C03660=1168.556,292.806,-70.556,-176.920,7.929,148.636
C03661=1168.552,293.053,-70.586,-176.917,7.932,148.636
C03662=1168.547,293.302,-70.616,-176.914,7.935,148.636
C03663=1168.544,293.551,-70.646,-176.912,7.938,148.636
C03664=1168.540,293.798,-70.676,-176.909,7.941,148.636
C03665=1168.535,294.047,-70.706,-176.907,7.944,148.636
C03666=1168.531,294.295,-70.736,-176.904,7.947,148.636
C03667=1168.527,294.543,-70.765,-176.902,7.950,148.636
C03668=1168.522,294.791,-70.796,-176.899,7.953,148.636
C03669=1168.518,295.039,-70.826,-176.896,7.956,148.636
C03670=1168.514,295.287,-70.855,-176.894,7.958,148.636
C03671=1168.509,295.535,-70.886,-176.892,7.962,148.636
C03672=1168.505,295.784,-70.915,-176.889,7.965,148.636
C03673=1168.501,296.032,-70.946,-176.886,7.968,148.636
C03674=1168.497,296.281,-70.976,-176.884,7.971,148.637
C03675=1168.493,296.528,-71.006,-176.881,7.974,148.637
C03676=1168.488,296.776,-71.037,-176.878,7.977,148.637
C03677=1168.484,297.024,-71.066,-176.876,7.980,148.637
C03678=1168.480,297.272,-71.097,-176.873,7.983,148.637
C03679=1168.475,297.521,-71.127,-176.871,7.986,148.637
C03680=1168.471,297.769,-71.157,-176.868,7.989,148.637
C03681=1168.467,298.018,-71.187,-176.866,7.992,148.637
C03682=1168.463,298.265,-71.217,-176.863,7.995,148.637
C03683=1168.459,298.513,-71.248,-176.861,7.999,148.637
C03684=1168.455,298.761,-71.278,-176.858,8.002,148.637
C03685=1168.450,299.009,-71.308,-176.855,8.005,148.637
C03686=1168.446,299.257,-71.338,-176.853,8.008,148.637
C03687=1168.442,299.506,-71.369,-176.850,8.011,148.637
C03688=1168.438,299.754,-71.399,-176.847,8.014,148.637
C03689=1168.433,300.002,-71.430,-176.845,8.017,148.637
C03690=1168.429,300.250,-71.461,-176.842,8.020,148.637
C03691=1168.425,300.498,-71.490,-176.840,8.023,148.637
C03692=1168.420,300.747,-71.521,-176.837,8.026,148.637
C03693=1168.417,300.994,-71.551,-176.835,8.029,148.637
C03694=1168.412,301.242,-71.582,-176.832,8.032,148.637
C03695=1168.408,301.490,-71.612,-176.830,8.036,148.637
C03696=1168.403,301.739,-71.642,-176.827,8.039,148.637
C03697=1168.399,301.987,-71.673,-176.825,8.042,148.638
C03698=1168.395,302.235,-71.704,-176.822,8.045,148.638
C03699=1168.391,302.483,-71.734,-176.819,8.048,148.638
C03700=1168.387,302.731,-71.765,-176.817,8.051,148.638
C03701=1168.383,302.979,-71.796,-176.814,8.054,148.638
C03702=1168.378,303.227,-71.826,-176.811,8.057,148.638
C03703=1168.374,303.475,-71.856,-176.809,8.060,148.638
C03704=1168.369,303.723,-71.887,-176.806,8.063,148.638
C03705=1168.365,303.972,-71.918,-176.804,8.067,148.638
C03706=1168.362,304.220,-71.948,-176.801,8.070,148.638
C03707=1168.357,304.468,-71.979,-176.798,8.073,148.638
C03708=1168.352,304.716,-72.009,-176.796,8.076,148.638
C03709=1168.348,304.964,-72.041,-176.793,8.079,148.638
C03710=1168.344,305.212,-72.071,-176.791,8.082,148.638
C03711=1168.340,305.460,-72.102,-176.788,8.085,148.638
C03712=1168.336,305.709,-72.133,-176.786,8.088,148.638
C03713=1168.332,305.956,-72.163,-176.783,8.092,148.639
C03714=1168.327,306.204,-72.194,-176.780,8.095,148.639
C03715=1168.324,306.452,-72.225,-176.778,8.099,148.639
C03716=1168.319,306.700,-72.256,-176.775,8.102,148.639
C03717=1168.314,306.948,-72.287,-176.773,8.105,148.639
C03718=1168.311,307.196,-72.317,-176.770,8.108,148.639
C03719=1168.306,307.444,-72.348,-176.767,8.111,148.639
C03720=1168.302,307.692,-72.379,-176.765,8.114,148.639
C03721=1168.298,307.941,-72.410,-176.762,8.117,148.639
C03722=1168.293,308.189,-72.441,-176.760,8.120,148.639
C03723=1168.290,308.436,-72.472,-176.757,8.123,148.639
C03724=1168.286,308.685,-72.503,-176.755,8.127,148.639
C03725=1168.281,308.933,-72.534,-176.752,8.130,148.639
C03726=1168.276,309.181,-72.564,-176.750,8.133,148.640
C03727=1168.272,309.429,-72.596,-176.747,8.136,148.640
C03728=1168.268,309.677,-72.627,-176.744,8.139,148.639
C03729=1168.264,309.925,-72.658,-176.742,8.142,148.640
C03730=1168.260,310.173,-72.688,-176.739,8.145,148.640
C03731=1168.256,310.420,-72.720,-176.737,8.148,148.640
C03732=1168.252,310.669,-72.751,-176.734,8.151,148.640
C03733=1168.247,310.917,-72.782,-176.732,8.155,148.640
C03734=1168.244,311.165,-72.814,-176.729,8.158,148.640
C03735=1168.239,311.413,-72.844,-176.727,8.161,148.640
C03736=1168.235,311.662,-72.875,-176.724,8.165,148.640
C03737=1168.231,311.909,-72.907,-176.721,8.168,148.640
C03738=1168.226,312.157,-72.938,-176.719,8.171,148.640
C03739=1168.222,312.405,-72.969,-176.716,8.174,148.641
C03740=1168.218,312.653,-73.000,-176.714,8.177,148.641
C03741=1168.214,312.901,-73.031,-176.711,8.181,148.641
C03742=1168.209,313.149,-73.063,-176.709,8.184,148.641
C03743=1168.205,313.397,-73.094,-176.706,8.187,148.641
C03744=1168.201,313.674,-73.129,-176.704,8.190,148.641
C03745=1168.196,313.951,-73.164,-176.701,8.194,148.641
C03746=1168.191,314.228,-73.198,-176.698,8.198,148.641
C03747=1168.187,314.506,-73.234,-176.695,8.201,148.641
C03748=1168.182,314.753,-73.266,-176.692,8.204,148.641
C03749=1168.178,315.002,-73.297,-176.690,8.207,148.642
C03750=1168.174,315.249,-73.328,-176.687,8.210,148.642
C03751=1168.170,315.498,-73.359,-176.685,8.214,148.642
C03752=1168.166,315.745,-73.391,-176.682,8.217,148.642
C03753=1168.162,315.993,-73.423,-176.680,8.221,148.642
C03754=1168.157,316.241,-73.453,-176.677,8.224,148.642
C03755=1168.154,316.489,-73.485,-176.675,8.227,148.642
C03756=1168.149,316.737,-73.516,-176.672,8.230,148.642
C03757=1168.145,316.985,-73.548,-176.670,8.233,148.642
C03758=1168.141,317.232,-73.579,-176.667,8.236,148.642
C03759=1168.136,317.481,-73.611,-176.664,8.240,148.643
C03760=1168.132,317.729,-73.643,-176.662,8.242,148.642
C03761=1168.128,317.977,-73.674,-176.659,8.246,148.643
C03762=1168.125,318.225,-73.706,-176.657,8.249,148.643
C03763=1168.120,318.473,-73.737,-176.654,8.252,148.643
C03764=1168.116,318.721,-73.769,-176.652,8.256,148.643
C03765=1168.111,318.968,-73.801,-176.649,8.259,148.643
C03766=1168.108,319.216,-73.833,-176.647,8.262,148.643
C03767=1168.104,319.465,-73.864,-176.644,8.265,148.643
C03768=1168.099,319.712,-73.895,-176.642,8.269,148.643
C03769=1168.096,319.961,-73.927,-176.639,8.272,148.644
C03770=1168.091,320.208,-73.959,-176.637,8.275,148.644
C03771=1168.087,320.456,-73.991,-176.634,8.278,148.644
C03772=1168.083,320.704,-74.023,-176.631,8.281,148.644
C03773=1168.079,320.952,-74.054,-176.629,8.285,148.644
C03774=1168.074,321.201,-74.086,-176.626,8.289,148.644
C03775=1168.070,321.449,-74.118,-176.624,8.292,148.644
C03776=1168.066,321.696,-74.149,-176.621,8.295,148.644
C03777=1168.062,321.944,-74.181,-176.619,8.298,148.644
C03778=1168.058,322.192,-74.214,-176.616,8.301,148.645
C03779=1168.054,322.440,-74.245,-176.614,8.305,148.645
C03780=1168.050,322.688,-74.277,-176.611,8.308,148.645
C03781=1168.045,322.936,-74.310,-176.609,8.311,148.645
C03782=1168.041,323.183,-74.341,-176.606,8.315,148.645
C03783=1168.037,323.431,-74.373,-176.603,8.318,148.645
C03784=1168.033,323.680,-74.405,-176.601,8.321,148.645
C03785=1168.029,323.927,-74.437,-176.598,8.324,148.645
C03786=1168.025,324.175,-74.469,-176.596,8.327,148.646
C03787=1168.021,324.424,-74.501,-176.594,8.331,148.646
C03788=1168.017,324.672,-74.533,-176.591,8.334,148.646
C03789=1168.013,324.919,-74.564,-176.589,8.337,148.646
C03790=1168.008,325.167,-74.597,-176.586,8.341,148.646
C03791=1168.004,325.415,-74.629,-176.583,8.344,148.646
C03792=1168.000,325.662,-74.661,-176.581,8.347,148.646
C03793=1167.996,325.910,-74.693,-176.579,8.351,148.647
C03794=1167.992,326.158,-74.725,-176.576,8.354,148.647
C03795=1167.988,326.407,-74.758,-176.574,8.357,148.647
C03796=1167.983,326.654,-74.789,-176.571,8.360,148.647
C03797=1167.979,326.902,-74.822,-176.569,8.363,148.647
C03798=1167.976,327.150,-74.854,-176.566,8.367,148.647
C03799=1167.971,327.398,-74.887,-176.563,8.371,148.648
C03800=1167.967,327.646,-74.918,-176.561,8.374,148.648
C03801=1167.962,327.894,-74.950,-176.558,8.377,148.648
C03802=1167.959,328.141,-74.983,-176.556,8.380,148.648
C03803=1167.955,328.390,-75.015,-176.554,8.384,148.648
C03804=1167.951,328.638,-75.047,-176.551,8.387,148.648
C03805=1167.946,328.885,-75.080,-176.548,8.391,148.648
C03806=1167.942,329.133,-75.112,-176.546,8.394,148.649
C03807=1167.938,329.381,-75.144,-176.543,8.397,148.649
C03808=1167.935,329.629,-75.177,-176.541,8.400,148.649
C03809=1167.930,329.877,-75.209,-176.539,8.404,148.649
C03810=1167.926,330.125,-75.242,-176.536,8.407,148.649
C03811=1167.922,330.372,-75.274,-176.533,8.411,148.649
C03812=1167.917,330.620,-75.306,-176.531,8.414,148.649
C03813=1167.914,330.868,-75.338,-176.528,8.417,148.650
C03814=1167.909,331.116,-75.371,-176.526,8.421,148.650
C03815=1167.905,331.364,-75.404,-176.523,8.423,148.650
C03816=1167.902,331.612,-75.436,-176.521,8.427,148.650
C03817=1167.897,331.859,-75.469,-176.518,8.431,148.650
C03818=1167.892,332.107,-75.502,-176.516,8.434,148.650
C03819=1167.889,332.355,-75.534,-176.513,8.437,148.650
C03820=1167.885,332.603,-75.567,-176.511,8.440,148.651
C03821=1167.880,332.851,-75.599,-176.509,8.444,148.651
C03822=1167.877,333.099,-75.632,-176.506,8.447,148.651
C03823=1167.872,333.347,-75.664,-176.504,8.451,148.651
C03824=1167.868,333.595,-75.697,-176.501,8.454,148.651
C03825=1167.864,333.842,-75.729,-176.498,8.457,148.652
C03826=1167.860,334.090,-75.762,-176.496,8.461,148.652
C03827=1167.856,334.338,-75.795,-176.494,8.464,148.652
C03828=1167.852,334.586,-75.827,-176.491,8.468,148.652
C03829=1167.848,334.833,-75.860,-176.488,8.471,148.652
C03830=1167.844,335.081,-75.893,-176.486,8.474,148.652
C03831=1167.839,335.329,-75.926,-176.484,8.478,148.653
C03832=1167.836,335.577,-75.958,-176.481,8.481,148.653
C03833=1167.832,335.825,-75.991,-176.479,8.484,148.653
C03834=1167.827,336.073,-76.024,-176.476,8.488,148.653
C03835=1167.823,336.321,-76.057,-176.474,8.491,148.653
C03836=1167.819,336.568,-76.090,-176.471,8.495,148.653
C03837=1167.815,336.816,-76.123,-176.469,8.498,148.654
C03838=1167.811,337.064,-76.155,-176.467,8.501,148.654
C03839=1167.807,337.312,-76.188,-176.464,8.505,148.654
C03840=1167.803,337.560,-76.221,-176.462,8.509,148.654
C03841=1167.799,337.807,-76.255,-176.459,8.512,148.654
C03842=1167.794,338.055,-76.288,-176.457,8.515,148.655
C03843=1167.791,338.303,-76.320,-176.454,8.518,148.655
C03844=1167.787,338.551,-76.353,-176.451,8.522,148.655
C03845=1167.782,338.799,-76.386,-176.449,8.526,148.655
C03846=1167.778,339.046,-76.419,-176.447,8.529,148.655
C03847=1167.774,339.294,-76.452,-176.445,8.532,148.656
C03848=1167.770,339.574,-76.490,-176.442,8.536,148.656
C03849=1167.764,339.853,-76.527,-176.438,8.540,148.656
C03850=1167.760,340.132,-76.563,-176.435,8.544,148.656
C03851=1167.756,340.412,-76.601,-176.433,8.548,148.656
C03852=1167.751,340.660,-76.634,-176.430,8.552,148.657
C03853=1167.747,340.907,-76.667,-176.428,8.555,148.657
C03854=1167.743,341.155,-76.700,-176.426,8.558,148.657
C03855=1167.739,341.403,-76.733,-176.423,8.562,148.657
C03856=1167.735,341.651,-76.766,-176.421,8.565,148.658
C03857=1167.731,341.898,-76.800,-176.418,8.569,148.658
C03858=1167.727,342.146,-76.833,-176.416,8.572,148.658
C03859=1167.723,342.394,-76.866,-176.414,8.576,148.658
C03860=1167.719,342.641,-76.900,-176.411,8.579,148.658
C03861=1167.715,342.889,-76.933,-176.409,8.583,148.659
C03862=1167.711,343.137,-76.966,-176.406,8.586,148.659
C03863=1167.707,343.385,-77.000,-176.404,8.590,148.659
C03864=1167.703,343.633,-77.033,-176.402,8.593,148.659
C03865=1167.699,343.880,-77.066,-176.399,8.597,148.660
C03866=1167.694,344.128,-77.099,-176.397,8.600,148.660
C03867=1167.690,344.376,-77.133,-176.394,8.604,148.660
C03868=1167.686,344.623,-77.167,-176.392,8.607,148.660
C03869=1167.682,344.871,-77.200,-176.389,8.611,148.660
C03870=1167.678,345.119,-77.233,-176.387,8.614,148.661
C03871=1167.674,345.367,-77.267,-176.385,8.618,148.661
C03872=1167.670,345.615,-77.300,-176.382,8.621,148.661
C03873=1167.666,345.862,-77.334,-176.379,8.625,148.661
C03874=1167.662,346.110,-77.367,-176.377,8.628,148.662
C03875=1167.657,346.358,-77.400,-176.375,8.632,148.662
C03876=1167.653,346.605,-77.434,-176.373,8.635,148.662
C03877=1167.650,346.853,-77.468,-176.370,8.639,148.662
C03878=1167.645,347.101,-77.501,-176.367,8.642,148.662
C03879=1167.641,347.349,-77.534,-176.365,8.646,148.663
C03880=1167.637,347.596,-77.568,-176.362,8.650,148.663
C03881=1167.633,347.844,-77.602,-176.360,8.653,148.663
C03882=1167.629,348.092,-77.636,-176.358,8.656,148.663
C03883=1167.625,348.339,-77.669,-176.355,8.660,148.664
C03884=1167.621,348.587,-77.702,-176.352,8.664,148.664
C03885=1167.617,348.834,-77.736,-176.350,8.667,148.664
C03886=1167.612,349.082,-77.770,-176.348,8.670,148.664
C03887=1167.609,349.330,-77.804,-176.346,8.674,148.665
C03888=1167.605,349.578,-77.837,-176.343,8.678,148.665
C03889=1167.601,349.825,-77.871,-176.341,8.681,148.665
C03890=1167.596,350.073,-77.905,-176.339,8.685,148.665
C03891=1167.593,350.321,-77.939,-176.336,8.689,148.666
C03892=1167.589,350.568,-77.972,-176.333,8.692,148.666
C03893=1167.584,350.816,-78.007,-176.331,8.695,148.666
C03894=1167.580,351.064,-78.040,-176.329,8.699,148.666
C03895=1167.577,351.311,-78.074,-176.326,8.703,148.667
C03896=1167.572,351.559,-78.108,-176.324,8.706,148.667
C03897=1167.568,351.807,-78.142,-176.322,8.710,148.667
C03898=1167.564,352.054,-78.175,-176.319,8.714,148.667
C03899=1167.560,352.302,-78.210,-176.317,8.717,148.668
C03900=1167.556,352.550,-78.244,-176.314,8.720,148.668
C03901=1167.552,352.797,-78.277,-176.312,8.725,148.668
C03902=1167.548,353.045,-78.312,-176.310,8.728,148.669
C03903=1167.544,353.292,-78.346,-176.307,8.731,148.669
C03904=1167.540,353.540,-78.379,-176.305,8.736,148.669
C03905=1167.536,353.788,-78.414,-176.302,8.739,148.669
C03906=1167.532,354.035,-78.447,-176.300,8.742,148.670
C03907=1167.528,354.283,-78.481,-176.298,8.746,148.670
C03908=1167.524,354.531,-78.515,-176.295,8.750,148.670
C03909=1167.521,354.778,-78.549,-176.293,8.753,148.670
C03910=1167.516,355.026,-78.584,-176.291,8.757,148.671
C03911=1167.512,355.274,-78.617,-176.288,8.761,148.671
C03912=1167.508,355.522,-78.652,-176.286,8.764,148.671
C03913=1167.504,355.769,-78.686,-176.284,8.768,148.671
C03914=1167.500,356.017,-78.720,-176.281,8.772,148.672
C03915=1167.496,356.264,-78.754,-176.279,8.775,148.672
C03916=1167.492,356.511,-78.789,-176.277,8.779,148.672
C03917=1167.488,356.760,-78.822,-176.274,8.783,148.673
C03918=1167.484,357.007,-78.857,-176.272,8.786,148.673
C03919=1167.480,357.255,-78.891,-176.270,8.790,148.673
C03920=1167.476,357.502,-78.925,-176.267,8.794,148.674
C03921=1167.472,357.750,-78.959,-176.265,8.797,148.674
C03922=1167.468,357.998,-78.994,-176.262,8.801,148.674
C03923=1167.464,358.245,-79.028,-176.260,8.805,148.674
C03924=1167.460,358.493,-79.063,-176.258,8.808,148.675
C03925=1167.456,358.740,-79.097,-176.255,8.812,148.675
C03926=1167.452,358.988,-79.132,-176.253,8.816,148.675
C03927=1167.448,359.236,-79.166,-176.251,8.819,148.676
C03928=1167.444,359.483,-79.200,-176.248,8.823,148.676
C03929=1167.440,359.731,-79.235,-176.246,8.827,148.676
C03930=1167.436,359.978,-79.269,-176.244,8.830,148.677
C03931=1167.432,360.226,-79.303,-176.241,8.834,148.677
C03932=1167.428,360.473,-79.338,-176.239,8.838,148.677
C03933=1167.424,360.721,-79.372,-176.236,8.842,148.678
C03934=1167.420,360.969,-79.407,-176.235,8.846,148.678
C03935=1167.416,361.217,-79.441,-176.232,8.849,148.678
C03936=1167.412,361.463,-79.476,-176.230,8.854,148.679
C03937=1167.408,361.711,-79.511,-176.228,8.857,148.679
C03938=1167.404,361.959,-79.545,-176.226,8.860,148.679
C03939=1167.401,362.207,-79.580,-176.223,8.865,148.680
C03940=1167.396,362.454,-79.614,-176.221,8.868,148.680
C03941=1167.392,362.702,-79.649,-176.219,8.871,148.680
C03942=1167.388,362.949,-79.683,-176.216,8.876,148.681
C03943=1167.385,363.197,-79.718,-176.214,8.879,148.681
C03944=1167.380,363.444,-79.753,-176.212,8.884,148.682
C03945=1167.377,363.692,-79.787,-176.209,8.887,148.682
C03946=1167.372,363.939,-79.822,-176.207,8.890,148.682
C03947=1167.368,364.187,-79.857,-176.205,8.895,148.683
C03948=1167.365,364.435,-79.892,-176.203,8.898,148.683
C03949=1167.361,364.682,-79.926,-176.201,8.902,148.683
C03950=1167.357,364.930,-79.961,-176.198,8.906,148.684
C03951=1167.352,365.177,-79.996,-176.197,8.910,148.684
C03952=1167.348,365.459,-80.036,-176.194,8.914,148.685
C03953=1167.344,365.742,-80.075,-176.191,8.918,148.685
C03954=1167.340,366.024,-80.115,-176.189,8.923,148.685
C03955=1167.335,366.306,-80.155,-176.187,8.926,148.686
C03956=1167.331,366.554,-80.189,-176.184,8.931,148.686
C03957=1167.326,366.801,-80.225,-176.183,8.934,148.687
C03958=1167.323,367.049,-80.260,-176.181,8.938,148.687
C03959=1167.319,367.296,-80.295,-176.178,8.942,148.688
C03960=1167.314,367.544,-80.330,-176.177,8.946,148.688
C03961=1167.311,367.792,-80.364,-176.174,8.949,148.688
C03962=1167.307,368.038,-80.399,-176.172,8.953,148.689
C03963=1167.303,368.286,-80.434,-176.170,8.957,148.689
C03964=1167.299,368.534,-80.469,-176.168,8.961,148.690
C03965=1167.295,368.781,-80.504,-176.167,8.965,148.690
C03966=1167.291,369.029,-80.539,-176.165,8.968,148.691
C03967=1167.287,369.276,-80.575,-176.163,8.972,148.691
C03968=1167.283,369.524,-80.609,-176.161,8.977,148.692
C03969=1167.279,369.771,-80.645,-176.159,8.980,148.692
C03970=1167.275,370.019,-80.680,-176.157,8.984,148.692
C03971=1167.271,370.266,-80.715,-176.155,8.987,148.693
C03972=1167.267,370.514,-80.750,-176.154,8.991,148.694
C03973=1167.263,370.762,-80.785,-176.152,8.995,148.694
C03974=1167.259,371.009,-80.820,-176.150,8.998,148.694
C03975=1167.255,371.257,-80.855,-176.147,9.003,148.695
C03976=1167.251,371.504,-80.891,-176.146,9.007,148.696
C03977=1167.247,371.751,-80.926,-176.144,9.010,148.696
C03978=1167.243,371.999,-80.962,-176.142,9.014,148.696
C03979=1167.239,372.247,-80.996,-176.141,9.018,148.697
C03980=1167.235,372.494,-81.032,-176.139,9.021,148.697
C03981=1167.231,372.741,-81.067,-176.138,9.025,148.698
C03982=1167.227,372.989,-81.102,-176.136,9.029,148.698
C03983=1167.224,373.237,-81.138,-176.134,9.033,148.699
C03984=1167.220,373.483,-81.173,-176.132,9.037,148.700
C03985=1167.216,373.731,-81.208,-176.131,9.040,148.700
C03986=1167.212,373.979,-81.243,-176.130,9.044,148.701
C03987=1167.208,374.226,-81.278,-176.128,9.048,148.701
C03988=1167.204,374.473,-81.314,-176.126,9.052,148.702
C03989=1167.200,374.721,-81.349,-176.125,9.056,148.702
C03990=1167.197,374.968,-81.385,-176.123,9.059,148.703
C03991=1167.192,375.215,-81.420,-176.122,9.062,148.703
C03992=1167.188,375.463,-81.455,-176.121,9.066,148.704
C03993=1167.184,375.711,-81.491,-176.119,9.070,148.705
C03994=1167.180,375.959,-81.527,-176.117,9.074,148.705
C03995=1167.176,376.205,-81.562,-176.116,9.078,148.706
C03996=1167.172,376.453,-81.597,-176.115,9.082,148.706
C03997=1167.169,376.700,-81.633,-176.114,9.085,148.707
C03998=1167.165,376.948,-81.668,-176.112,9.089,148.708
C03999=1167.161,377.195,-81.704,-176.111,9.093,148.708
C04000=1167.156,377.442,-81.740,-176.109,9.096,148.709
C04001=1167.153,377.690,-81.775,-176.109,9.100,148.709
C04002=1167.149,377.938,-81.811,-176.107,9.103,148.710
C04003=1167.145,378.185,-81.846,-176.106,9.107,148.711
C04004=1167.141,378.432,-81.882,-176.105,9.110,148.711
C04005=1167.137,378.680,-81.918,-176.103,9.114,148.712
C04006=1167.133,378.927,-81.953,-176.103,9.118,148.713
C04007=1167.129,379.175,-81.989,-176.102,9.122,148.713
C04008=1167.126,379.422,-82.024,-176.100,9.126,148.714
C04009=1167.122,379.670,-82.060,-176.099,9.129,148.714
C04010=1167.117,379.917,-82.096,-176.098,9.133,148.715
C04011=1167.114,380.164,-82.131,-176.098,9.136,148.716
C04012=1167.110,380.412,-82.167,-176.096,9.140,148.717
C04013=1167.106,380.659,-82.202,-176.095,9.143,148.717
C04014=1167.102,380.907,-82.238,-176.094,9.147,148.718
C04015=1167.098,381.154,-82.274,-176.093,9.150,148.718
C04016=1167.094,381.401,-82.309,-176.093,9.154,148.719
C04017=1167.090,381.649,-82.345,-176.092,9.158,148.720
C04018=1167.086,381.897,-82.381,-176.091,9.161,148.721
C04019=1167.082,382.144,-82.417,-176.090,9.164,148.721
C04020=1167.079,382.391,-82.453,-176.089,9.168,148.722
C04021=1167.074,382.639,-82.489,-176.088,9.171,148.723
C04022=1167.070,382.886,-82.524,-176.088,9.175,148.723
C04023=1167.066,383.133,-82.560,-176.088,9.178,148.724
C04024=1167.063,383.381,-82.595,-176.086,9.182,148.725
C04025=1167.059,383.628,-82.632,-176.086,9.185,148.726
C04026=1167.055,383.875,-82.668,-176.085,9.188,148.726
C04027=1167.051,384.123,-82.703,-176.084,9.192,148.727
C04028=1167.047,384.371,-82.739,-176.084,9.195,148.728
C04029=1167.043,384.618,-82.775,-176.084,9.199,148.728
C04030=1167.039,384.864,-82.811,-176.083,9.202,148.729
C04031=1167.035,385.112,-82.847,-176.082,9.205,148.730
C04032=1167.031,385.360,-82.882,-176.082,9.209,148.731
C04033=1167.028,385.607,-82.918,-176.081,9.212,148.731
C04034=1167.024,385.854,-82.955,-176.081,9.215,148.732
C04035=1167.020,386.102,-82.990,-176.081,9.219,148.733
C04036=1167.016,386.349,-83.026,-176.080,9.222,148.734
C04037=1167.012,386.597,-83.062,-176.080,9.224,148.734
C04038=1167.008,386.844,-83.098,-176.079,9.228,148.735
C04039=1167.004,387.092,-83.134,-176.079,9.231,148.736
C04040=1167.000,387.339,-83.170,-176.079,9.235,148.736
C04041=1166.996,387.585,-83.206,-176.079,9.237,148.737
C04042=1166.992,387.833,-83.242,-176.078,9.240,148.738
C04043=1166.988,388.081,-83.278,-176.078,9.244,148.739
C04044=1166.985,388.328,-83.314,-176.078,9.246,148.739
C04045=1166.981,388.576,-83.350,-176.078,9.250,148.740
C04046=1166.977,388.823,-83.386,-176.078,9.253,148.741
C04047=1166.973,389.070,-83.422,-176.078,9.256,148.742
C04048=1166.969,389.318,-83.458,-176.078,9.259,148.743
C04049=1166.966,389.565,-83.493,-176.077,9.262,148.743
C04050=1166.961,389.812,-83.530,-176.078,9.265,148.744
C04051=1166.958,390.060,-83.566,-176.077,9.268,148.745
C04052=1166.953,390.308,-83.602,-176.077,9.271,148.746
C04053=1166.950,390.555,-83.638,-176.077,9.274,148.746
C04054=1166.945,390.802,-83.674,-176.078,9.277,148.747
C04055=1166.942,391.049,-83.710,-176.078,9.279,148.748
C04056=1166.937,391.334,-83.752,-176.077,9.283,148.749
C04057=1166.933,391.619,-83.793,-176.078,9.286,148.750
C04058=1166.929,391.904,-83.835,-176.078,9.289,148.751
C04059=1166.924,392.189,-83.876,-176.078,9.292,148.751
C04060=1166.920,392.437,-83.913,-176.078,9.296,148.752
C04061=1166.916,392.684,-83.948,-176.078,9.298,148.753
C04062=1166.912,392.931,-83.985,-176.078,9.301,148.754
C04063=1166.908,393.179,-84.021,-176.078,9.303,148.754
C04064=1166.904,393.427,-84.057,-176.079,9.306,148.755
C04065=1166.900,393.674,-84.093,-176.079,9.309,148.756
C04066=1166.897,393.921,-84.129,-176.079,9.311,148.757
C04067=1166.893,394.168,-84.166,-176.079,9.314,148.757
C04068=1166.889,394.416,-84.201,-176.080,9.316,148.758
C04069=1166.885,394.663,-84.238,-176.080,9.319,148.759
C04070=1166.881,394.910,-84.273,-176.080,9.322,148.760
C04071=1166.877,395.158,-84.310,-176.080,9.324,148.761
C04072=1166.873,395.405,-84.346,-176.081,9.327,148.761
C04073=1166.869,395.653,-84.382,-176.081,9.330,148.762
C04074=1166.866,395.900,-84.418,-176.081,9.332,148.763
C04075=1166.861,396.148,-84.454,-176.082,9.334,148.764
C04076=1166.858,396.395,-84.491,-176.082,9.337,148.764
C04077=1166.854,396.642,-84.527,-176.082,9.339,148.765
C04078=1166.850,396.889,-84.563,-176.082,9.342,148.766
C04079=1166.846,397.137,-84.599,-176.083,9.345,148.766
C04080=1166.842,397.384,-84.635,-176.083,9.346,148.767
C04081=1166.838,397.632,-84.672,-176.084,9.349,148.768
C04082=1166.835,397.879,-84.708,-176.084,9.352,148.769
C04083=1166.830,398.126,-84.744,-176.084,9.354,148.769
C04084=1166.827,398.373,-84.780,-176.085,9.356,148.770
C04085=1166.823,398.621,-84.816,-176.085,9.359,148.771
C04086=1166.819,398.868,-84.853,-176.085,9.361,148.771
C04087=1166.815,399.116,-84.889,-176.086,9.363,148.772
C04088=1166.811,399.363,-84.925,-176.086,9.366,148.773
C04089=1166.807,399.610,-84.961,-176.087,9.368,148.774
C04090=1166.804,399.857,-84.998,-176.087,9.370,148.774
C04091=1166.799,400.105,-85.034,-176.087,9.373,148.775
C04092=1166.795,400.352,-85.071,-176.088,9.374,148.776
C04093=1166.792,400.599,-85.107,-176.088,9.377,148.776
C04094=1166.787,400.847,-85.143,-176.088,9.380,148.777
C04095=1166.784,401.094,-85.179,-176.089,9.381,148.778
C04096=1166.780,401.342,-85.215,-176.089,9.384,148.778
C04097=1166.776,401.589,-85.252,-176.090,9.386,148.779
C04098=1166.772,401.836,-85.288,-176.090,9.388,148.780
C04099=1166.769,402.083,-85.324,-176.091,9.390,148.781
C04100=1166.764,402.331,-85.360,-176.091,9.392,148.781
C04101=1166.761,402.578,-85.396,-176.092,9.394,148.782
C04102=1166.756,402.826,-85.433,-176.092,9.397,148.783
C04103=1166.753,403.073,-85.469,-176.092,9.399,148.783
C04104=1166.749,403.320,-85.506,-176.093,9.400,148.784
C04105=1166.745,403.567,-85.541,-176.093,9.403,148.785
C04106=1166.741,403.815,-85.578,-176.094,9.405,148.785
C04107=1166.737,404.062,-85.614,-176.094,9.407,148.786
C04108=1166.733,404.309,-85.650,-176.095,9.409,148.787
C04109=1166.729,404.557,-85.687,-176.096,9.411,148.787
C04110=1166.726,404.804,-85.723,-176.096,9.413,148.788
C04111=1166.722,405.051,-85.760,-176.096,9.415,148.789
C04112=1166.718,405.299,-85.795,-176.097,9.418,148.789
C04113=1166.714,405.546,-85.832,-176.097,9.419,148.790
C04114=1166.710,405.793,-85.868,-176.098,9.421,148.790
C04115=1166.706,406.041,-85.905,-176.098,9.423,148.791
C04116=1166.702,406.288,-85.941,-176.098,9.425,148.792
C04117=1166.698,406.535,-85.977,-176.099,9.427,148.792
C04118=1166.694,406.782,-86.014,-176.099,9.429,148.793
C04119=1166.691,407.030,-86.049,-176.100,9.431,148.794
C04120=1166.686,407.277,-86.086,-176.100,9.433,148.794
C04121=1166.683,407.525,-86.122,-176.100,9.435,148.795
C04122=1166.679,407.772,-86.159,-176.101,9.437,148.796
C04123=1166.675,408.019,-86.195,-176.102,9.439,148.796
C04124=1166.671,408.266,-86.231,-176.102,9.440,148.797
C04125=1166.667,408.514,-86.268,-176.102,9.443,148.797
C04126=1166.663,408.761,-86.303,-176.103,9.444,148.798
C04127=1166.659,409.008,-86.340,-176.104,9.446,148.799
C04128=1166.656,409.255,-86.377,-176.103,9.448,148.799
C04129=1166.651,409.503,-86.413,-176.104,9.450,148.800
C04130=1166.647,409.750,-86.450,-176.105,9.452,148.801
C04131=1166.644,409.997,-86.486,-176.105,9.454,148.801
C04132=1166.639,410.245,-86.522,-176.105,9.456,148.802
C04133=1166.636,410.492,-86.558,-176.106,9.458,148.802
C04134=1166.632,410.740,-86.594,-176.107,9.459,148.803
C04135=1166.628,410.986,-86.631,-176.107,9.461,148.803
C04136=1166.624,411.234,-86.668,-176.107,9.463,148.804
C04137=1166.620,411.481,-86.704,-176.107,9.465,148.805
C04138=1166.617,411.728,-86.740,-176.108,9.467,148.805
C04139=1166.612,411.976,-86.777,-176.109,9.468,148.806
C04140=1166.609,412.223,-86.812,-176.108,9.471,148.806
C04141=1166.605,412.470,-86.849,-176.109,9.472,148.807
C04142=1166.601,412.717,-86.886,-176.109,9.474,148.808
C04143=1166.597,412.965,-86.922,-176.110,9.475,148.808
C04144=1166.593,413.212,-86.958,-176.110,9.478,148.809
C04145=1166.589,413.460,-86.994,-176.110,9.479,148.809
C04146=1166.586,413.708,-87.031,-176.111,9.481,148.810
C04147=1166.582,413.955,-87.068,-176.111,9.483,148.810
C04148=1166.578,414.202,-87.104,-176.112,9.484,148.811
C04149=1166.574,414.449,-87.140,-176.112,9.487,148.812
C04150=1166.570,414.696,-87.177,-176.113,9.488,148.812
C04151=1166.566,414.944,-87.213,-176.113,9.490,148.813
C04152=1166.562,415.191,-87.250,-176.114,9.492,148.813
C04153=1166.559,415.438,-87.286,-176.113,9.494,148.814
C04154=1166.557,415.685,-87.322,-176.114,9.496,148.815
C04155=1166.555,415.933,-87.358,-176.114,9.497,148.815
C04156=1166.554,416.247,-87.404,-176.115,9.499,148.816
C04157=1166.555,416.560,-87.449,-176.115,9.501,148.816
C04158=1166.556,416.874,-87.495,-176.116,9.503,148.817
C04159=1166.561,417.186,-87.540,-176.115,9.505,148.817
C04160=1166.140,417.187,-87.586,-176.119,9.516,148.821
C04161=1166.136,416.872,-87.540,-176.119,9.514,148.821
C04162=1166.133,416.556,-87.494,-176.118,9.512,148.820
C04163=1166.133,416.238,-87.448,-176.118,9.509,148.819
C04164=1166.133,415.922,-87.402,-176.117,9.508,148.819
C04165=1166.135,415.674,-87.366,-176.117,9.506,148.818
C04166=1166.138,415.427,-87.330,-176.117,9.505,148.818
C04167=1166.141,415.179,-87.293,-176.116,9.502,148.817
C04168=1166.144,414.932,-87.257,-176.116,9.501,148.816
C04169=1166.148,414.685,-87.220,-176.115,9.499,148.816
C04170=1166.153,414.437,-87.184,-176.115,9.498,148.815
C04171=1166.156,414.190,-87.147,-176.115,9.495,148.815
C04172=1166.160,413.943,-87.111,-176.115,9.494,148.814
C04173=1166.165,413.695,-87.074,-176.114,9.492,148.814
C04174=1166.168,413.449,-87.038,-176.114,9.490,148.813
C04175=1166.172,413.201,-87.001,-176.113,9.489,148.812
C04176=1166.176,412.954,-86.966,-176.113,9.486,148.812
C04177=1166.180,412.707,-86.929,-176.113,9.485,148.811
C04178=1166.184,412.459,-86.893,-176.112,9.483,148.811
C04179=1166.188,412.212,-86.856,-176.112,9.482,148.810
C04180=1166.192,411.965,-86.820,-176.112,9.479,148.809
C04181=1166.195,411.717,-86.784,-176.111,9.477,148.809
C04182=1166.200,411.470,-86.747,-176.111,9.476,148.808
C04183=1166.204,411.223,-86.710,-176.110,9.474,148.808
C04184=1166.207,410.975,-86.675,-176.109,9.472,148.807
C04185=1166.211,410.728,-86.638,-176.109,9.470,148.807
C04186=1166.215,410.481,-86.602,-176.109,9.468,148.806
C04187=1166.219,410.233,-86.566,-176.108,9.467,148.805
C04188=1166.223,409.986,-86.529,-176.108,9.465,148.805
C04189=1166.227,409.739,-86.492,-176.108,9.463,148.804
C04190=1166.231,409.492,-86.456,-176.107,9.461,148.803
C04191=1166.234,409.245,-86.420,-176.107,9.459,148.803
C04192=1166.239,408.997,-86.384,-176.106,9.458,148.802
C04193=1166.242,408.750,-86.348,-176.106,9.455,148.802
C04194=1166.246,408.503,-86.311,-176.105,9.453,148.801
C04195=1166.250,408.254,-86.274,-176.105,9.452,148.801
C04196=1166.253,408.007,-86.238,-176.105,9.449,148.800
C04197=1166.257,407.760,-86.201,-176.104,9.448,148.799
C04198=1166.261,407.513,-86.166,-176.103,9.446,148.799
C04199=1166.265,407.266,-86.129,-176.102,9.444,148.798
C04200=1166.269,407.018,-86.093,-176.103,9.442,148.797
C04201=1166.273,406.771,-86.056,-176.102,9.440,148.797
C04202=1166.277,406.524,-86.019,-176.101,9.438,148.796
C04203=1166.281,406.276,-85.984,-176.101,9.436,148.795
C04204=1166.285,406.029,-85.947,-176.101,9.434,148.795
C04205=1166.288,405.782,-85.911,-176.100,9.432,148.794
C04206=1166.293,405.534,-85.875,-176.100,9.430,148.793
C04207=1166.296,405.287,-85.838,-176.099,9.428,148.793
C04208=1166.300,405.040,-85.802,-176.099,9.426,148.792
C04209=1166.304,404.792,-85.765,-176.099,9.424,148.792
C04210=1166.308,404.545,-85.730,-176.098,9.422,148.791
C04211=1166.312,404.298,-85.693,-176.097,9.420,148.790
C04212=1166.316,404.050,-85.657,-176.097,9.418,148.790
C04213=1166.320,403.803,-85.621,-176.096,9.416,148.789
C04214=1166.323,403.556,-85.584,-176.096,9.414,148.788
C04215=1166.328,403.308,-85.548,-176.095,9.412,148.788
C04216=1166.331,403.061,-85.512,-176.095,9.410,148.787
C04217=1166.335,402.814,-85.476,-176.095,9.407,148.786
C04218=1166.340,402.566,-85.439,-176.094,9.406,148.785
C04219=1166.343,402.320,-85.403,-176.094,9.403,148.785
C04220=1166.347,402.072,-85.366,-176.093,9.401,148.784
C04221=1166.351,401.825,-85.330,-176.093,9.399,148.783
C04222=1166.355,401.577,-85.294,-176.092,9.397,148.783
C04223=1166.358,401.330,-85.258,-176.092,9.395,148.782
C04224=1166.363,401.082,-85.222,-176.091,9.393,148.781
C04225=1166.366,400.836,-85.185,-176.091,9.390,148.781
C04226=1166.371,400.588,-85.149,-176.090,9.388,148.780
C04227=1166.374,400.341,-85.113,-176.090,9.386,148.779
C04228=1166.378,400.093,-85.077,-176.089,9.384,148.778
C04229=1166.382,399.846,-85.041,-176.089,9.381,148.778
C04230=1166.386,399.599,-85.004,-176.089,9.379,148.777
C04231=1166.389,399.351,-84.968,-176.088,9.377,148.776
C04232=1166.394,399.104,-84.931,-176.088,9.374,148.776
C04233=1166.398,398.856,-84.895,-176.088,9.372,148.775
C04234=1166.401,398.610,-84.859,-176.087,9.370,148.774
C04235=1166.406,398.362,-84.823,-176.087,9.368,148.774
C04236=1166.409,398.115,-84.786,-176.087,9.365,148.773
C04237=1166.413,397.867,-84.750,-176.086,9.363,148.772
C04238=1166.417,397.620,-84.714,-176.086,9.360,148.771
C04239=1166.421,397.372,-84.678,-176.086,9.358,148.771
C04240=1166.425,397.126,-84.642,-176.085,9.356,148.770
C04241=1166.429,396.878,-84.606,-176.084,9.353,148.769
C04242=1166.432,396.631,-84.569,-176.084,9.351,148.768
C04243=1166.437,396.383,-84.533,-176.084,9.348,148.768
C04244=1166.440,396.136,-84.497,-176.084,9.345,148.767
C04245=1166.444,395.888,-84.461,-176.083,9.344,148.766
C04246=1166.448,395.641,-84.424,-176.083,9.341,148.765
C04247=1166.452,395.394,-84.388,-176.082,9.338,148.765
C04248=1166.456,395.147,-84.352,-176.082,9.336,148.764
C04249=1166.460,394.899,-84.316,-176.082,9.333,148.763
C04250=1166.463,394.652,-84.280,-176.082,9.331,148.763
C04251=1166.468,394.404,-84.244,-176.081,9.328,148.762
C04252=1166.472,394.158,-84.208,-176.081,9.325,148.761
C04253=1166.476,393.910,-84.171,-176.081,9.323,148.760
C04254=1166.480,393.663,-84.136,-176.081,9.320,148.760
C04255=1166.484,393.416,-84.099,-176.080,9.317,148.759
C04256=1166.488,393.168,-84.064,-176.080,9.315,148.758
C04257=1166.491,392.921,-84.027,-176.080,9.312,148.757
C04258=1166.495,392.673,-83.991,-176.080,9.309,148.756
C04259=1166.499,392.426,-83.955,-176.080,9.307,148.756
C04260=1166.503,392.179,-83.919,-176.079,9.304,148.755
C04261=1166.507,391.894,-83.877,-176.080,9.301,148.754
C04262=1166.512,391.609,-83.836,-176.080,9.297,148.753
C04263=1166.516,391.323,-83.794,-176.079,9.294,148.752
C04264=1166.521,391.038,-83.752,-176.080,9.291,148.751
C04265=1166.525,390.791,-83.716,-176.079,9.288,148.751
C04266=1166.528,390.544,-83.680,-176.079,9.285,148.750
C04267=1166.533,390.296,-83.644,-176.079,9.282,148.749
C04268=1166.537,390.048,-83.608,-176.079,9.279,148.748
C04269=1166.540,389.802,-83.572,-176.079,9.277,148.748
C04270=1166.544,389.554,-83.536,-176.079,9.273,148.747
C04271=1166.548,389.307,-83.500,-176.079,9.271,148.746
C04272=1166.552,389.059,-83.464,-176.079,9.267,148.745
C04273=1166.556,388.811,-83.428,-176.079,9.264,148.744
C04274=1166.559,388.565,-83.392,-176.080,9.261,148.744
C04275=1166.563,388.317,-83.356,-176.079,9.258,148.743
C04276=1166.567,388.069,-83.320,-176.080,9.255,148.742
C04277=1166.571,387.822,-83.283,-176.080,9.252,148.741
C04278=1166.575,387.575,-83.248,-176.080,9.249,148.741
C04279=1166.579,387.327,-83.212,-176.081,9.246,148.740
C04280=1166.583,387.081,-83.176,-176.081,9.242,148.739
C04281=1166.587,386.833,-83.140,-176.081,9.239,148.738
C04282=1166.591,386.585,-83.104,-176.081,9.236,148.738
C04283=1166.595,386.338,-83.068,-176.082,9.233,148.737
C04284=1166.598,386.091,-83.032,-176.082,9.230,148.736
C04285=1166.603,385.843,-82.996,-176.082,9.226,148.735
C04286=1166.606,385.596,-82.960,-176.083,9.223,148.735
C04287=1166.610,385.349,-82.924,-176.083,9.219,148.734
C04288=1166.614,385.101,-82.888,-176.084,9.216,148.733
C04289=1166.618,384.853,-82.852,-176.085,9.213,148.732
C04290=1166.622,384.607,-82.817,-176.085,9.210,148.732
C04291=1166.626,384.359,-82.780,-176.085,9.206,148.731
C04292=1166.630,384.112,-82.745,-176.086,9.203,148.730
C04293=1166.633,383.864,-82.709,-176.087,9.200,148.730
C04294=1166.638,383.617,-82.673,-176.087,9.196,148.729
C04295=1166.642,383.369,-82.638,-176.088,9.193,148.728
C04296=1166.645,383.122,-82.601,-176.088,9.190,148.727
C04297=1166.649,382.874,-82.565,-176.089,9.186,148.727
C04298=1166.653,382.627,-82.530,-176.090,9.183,148.726
C04299=1166.657,382.380,-82.494,-176.091,9.179,148.725
C04300=1166.662,382.132,-82.458,-176.092,9.175,148.724
C04301=1166.665,381.885,-82.422,-176.093,9.172,148.724
C04302=1166.669,381.638,-82.387,-176.093,9.168,148.723
C04303=1166.672,381.390,-82.351,-176.094,9.165,148.723
C04304=1166.677,381.143,-82.315,-176.095,9.161,148.722
C04305=1166.681,380.896,-82.280,-176.096,9.158,148.721
C04306=1166.685,380.648,-82.244,-176.097,9.154,148.721
C04307=1166.689,380.401,-82.208,-176.098,9.151,148.720
C04308=1166.693,380.153,-82.172,-176.099,9.147,148.719
C04309=1166.696,379.906,-82.137,-176.100,9.144,148.719
C04310=1166.700,379.658,-82.101,-176.101,9.140,148.718
C04311=1166.705,379.411,-82.066,-176.102,9.136,148.717
C04312=1166.708,379.164,-82.029,-176.103,9.133,148.717
C04313=1166.712,378.917,-81.994,-176.105,9.129,148.716
C04314=1166.716,378.669,-81.958,-176.105,9.126,148.715
C04315=1166.719,378.422,-81.923,-176.106,9.121,148.715
C04316=1166.724,378.174,-81.886,-176.107,9.118,148.714
C04317=1166.728,377.927,-81.851,-176.109,9.114,148.713
C04318=1166.732,377.679,-81.816,-176.110,9.110,148.713
C04319=1166.735,377.432,-81.780,-176.112,9.107,148.712
C04320=1166.739,377.184,-81.745,-176.112,9.103,148.711
C04321=1166.744,376.937,-81.710,-176.114,9.100,148.711
C04322=1166.748,376.689,-81.674,-176.115,9.096,148.710
C04323=1166.752,376.442,-81.638,-176.117,9.092,148.710
C04324=1166.755,376.194,-81.603,-176.118,9.089,148.709
C04325=1166.759,375.947,-81.567,-176.119,9.085,148.709
C04326=1166.763,375.700,-81.532,-176.121,9.081,148.708
C04327=1166.767,375.452,-81.497,-176.122,9.077,148.707
C04328=1166.771,375.205,-81.461,-176.124,9.073,148.707
C04329=1166.775,374.957,-81.425,-176.125,9.069,148.706
C04330=1166.780,374.710,-81.391,-176.127,9.066,148.706
C04331=1166.783,374.462,-81.355,-176.128,9.062,148.705
C04332=1166.787,374.215,-81.319,-176.129,9.059,148.704
C04333=1166.791,373.967,-81.284,-176.131,9.055,148.704
C04334=1166.795,373.720,-81.249,-176.133,9.051,148.703
C04335=1166.798,373.473,-81.213,-176.134,9.048,148.703
C04336=1166.802,373.225,-81.178,-176.136,9.044,148.702
C04337=1166.806,372.977,-81.143,-176.138,9.040,148.702
C04338=1166.810,372.730,-81.108,-176.139,9.036,148.701
C04339=1166.814,372.483,-81.072,-176.141,9.033,148.701
C04340=1166.818,372.235,-81.037,-176.143,9.028,148.700
C04341=1166.822,371.988,-81.002,-176.145,9.024,148.700
C04342=1166.826,371.741,-80.966,-176.146,9.020,148.699
C04343=1166.830,371.492,-80.932,-176.148,9.017,148.699
C04344=1166.834,371.246,-80.896,-176.150,9.013,148.698
C04345=1166.838,370.998,-80.861,-176.151,9.009,148.698
C04346=1166.842,370.750,-80.826,-176.153,9.006,148.697
C04347=1166.846,370.503,-80.791,-176.155,9.002,148.697
C04348=1166.850,370.256,-80.755,-176.157,8.999,148.696
C04349=1166.854,370.008,-80.721,-176.159,8.994,148.696
C04350=1166.858,369.761,-80.685,-176.161,8.990,148.695
C04351=1166.862,369.513,-80.650,-176.163,8.987,148.695
C04352=1166.866,369.265,-80.615,-176.164,8.983,148.694
C04353=1166.870,369.018,-80.580,-176.166,8.979,148.694
C04354=1166.874,368.770,-80.545,-176.169,8.975,148.694
C04355=1166.877,368.523,-80.509,-176.171,8.971,148.693
C04356=1166.882,368.275,-80.475,-176.172,8.968,148.693
C04357=1166.886,368.028,-80.439,-176.174,8.964,148.692
C04358=1166.890,367.780,-80.405,-176.177,8.960,148.692
C04359=1166.893,367.533,-80.370,-176.179,8.956,148.691
C04360=1166.897,367.285,-80.335,-176.180,8.953,148.691
C04361=1166.901,367.038,-80.300,-176.182,8.949,148.690
C04362=1166.905,366.790,-80.265,-176.185,8.945,148.690
C04363=1166.909,366.543,-80.230,-176.187,8.941,148.690
C04364=1166.914,366.295,-80.195,-176.189,8.938,148.689
C04365=1166.918,366.013,-80.155,-176.191,8.933,148.689
C04366=1166.922,365.731,-80.115,-176.194,8.929,148.688
C04367=1166.926,365.448,-80.076,-176.196,8.924,148.688
C04368=1166.931,365.167,-80.036,-176.199,8.920,148.687
C04369=1166.935,364.918,-80.001,-176.200,8.916,148.687
C04370=1166.939,364.670,-79.967,-176.203,8.912,148.687
C04371=1166.944,364.423,-79.931,-176.205,8.909,148.686
C04372=1166.947,364.176,-79.897,-176.207,8.905,148.686
C04373=1166.951,363.928,-79.863,-176.210,8.901,148.686
C04374=1166.955,363.681,-79.827,-176.212,8.897,148.685
C04375=1166.960,363.433,-79.793,-176.214,8.894,148.685
C04376=1166.963,363.186,-79.758,-176.217,8.890,148.685
C04377=1166.967,362.938,-79.724,-176.218,8.886,148.684
C04378=1166.971,362.691,-79.688,-176.221,8.883,148.684
C04379=1166.975,362.444,-79.654,-176.223,8.878,148.683
C04380=1166.979,362.195,-79.620,-176.225,8.875,148.683
C04381=1166.983,361.948,-79.585,-176.228,8.871,148.683
C04382=1166.987,361.700,-79.551,-176.230,8.867,148.682
C04383=1166.991,361.453,-79.516,-176.232,8.864,148.682
C04384=1166.995,361.205,-79.481,-176.235,8.859,148.682
C04385=1166.999,360.958,-79.447,-176.237,8.856,148.681
C04386=1167.003,360.710,-79.412,-176.239,8.853,148.681
C04387=1167.007,360.463,-79.378,-176.241,8.848,148.681
C04388=1167.010,360.215,-79.344,-176.244,8.845,148.680
C04389=1167.015,359.967,-79.309,-176.247,8.841,148.680
C04390=1167.019,359.719,-79.274,-176.248,8.837,148.680
C04391=1167.023,359.472,-79.240,-176.251,8.834,148.680
C04392=1167.027,359.224,-79.206,-176.253,8.829,148.679
C04393=1167.031,358.977,-79.172,-176.255,8.826,148.679
C04394=1167.035,358.729,-79.137,-176.258,8.823,148.679
C04395=1167.038,358.482,-79.103,-176.260,8.818,148.678
C04396=1167.043,358.234,-79.068,-176.262,8.815,148.678
C04397=1167.047,357.986,-79.034,-176.265,8.811,148.678
C04398=1167.051,357.739,-79.000,-176.267,8.807,148.677
C04399=1167.055,357.491,-78.965,-176.269,8.804,148.677
C04400=1167.059,357.244,-78.931,-176.272,8.800,148.677
C04401=1167.063,356.996,-78.896,-176.274,8.796,148.676
C04402=1167.066,356.749,-78.862,-176.276,8.793,148.676
C04403=1167.071,356.501,-78.828,-176.279,8.789,148.676
C04404=1167.074,356.253,-78.794,-176.282,8.786,148.676
C04405=1167.079,356.005,-78.760,-176.283,8.782,148.675
C04406=1167.083,355.758,-78.726,-176.286,8.778,148.675
C04407=1167.087,355.510,-78.691,-176.289,8.775,148.675
C04408=1167.091,355.263,-78.657,-176.290,8.771,148.674
C04409=1167.095,355.015,-78.623,-176.293,8.767,148.674
C04410=1167.099,354.767,-78.589,-176.296,8.764,148.674
C04411=1167.103,354.520,-78.555,-176.298,8.760,148.674
C04412=1167.107,354.272,-78.521,-176.301,8.756,148.673
C04413=1167.110,354.025,-78.487,-176.303,8.753,148.673
C04414=1167.115,353.777,-78.453,-176.305,8.749,148.673
C04415=1167.119,353.529,-78.419,-176.308,8.745,148.672
C04416=1167.122,353.282,-78.385,-176.310,8.742,148.672
C04417=1167.127,353.034,-78.350,-176.312,8.738,148.672
C04418=1167.131,352.786,-78.317,-176.315,8.734,148.672
C04419=1167.135,352.539,-78.282,-176.317,8.731,148.671
C04420=1167.139,352.291,-78.249,-176.319,8.728,148.671
C04421=1167.143,352.044,-78.215,-176.322,8.723,148.671
C04422=1167.147,351.796,-78.181,-176.325,8.720,148.671
C04423=1167.151,351.548,-78.147,-176.326,8.717,148.670
C04424=1167.155,351.301,-78.114,-176.329,8.713,148.670
C04425=1167.159,351.052,-78.079,-176.332,8.709,148.670
C04426=1167.163,350.805,-78.046,-176.334,8.706,148.669
C04427=1167.167,350.558,-78.012,-176.336,8.703,148.669
C04428=1167.172,350.310,-77.978,-176.339,8.698,148.669
C04429=1167.175,350.062,-77.944,-176.341,8.695,148.669
C04430=1167.179,349.814,-77.911,-176.343,8.692,148.668
C04431=1167.183,349.567,-77.877,-176.346,8.687,148.668
C04432=1167.188,349.319,-77.843,-176.348,8.684,148.668
C04433=1167.192,349.071,-77.810,-176.351,8.681,148.668
C04434=1167.195,348.824,-77.776,-176.353,8.678,148.667
C04435=1167.199,348.576,-77.742,-176.356,8.673,148.667
C04436=1167.204,348.328,-77.708,-176.358,8.670,148.667
C04437=1167.208,348.081,-77.675,-176.360,8.667,148.667
C04438=1167.211,347.833,-77.641,-176.363,8.663,148.667
C04439=1167.215,347.585,-77.607,-176.365,8.659,148.666
C04440=1167.220,347.337,-77.574,-176.368,8.656,148.666
C04441=1167.224,347.090,-77.540,-176.370,8.653,148.666
C04442=1167.228,346.842,-77.507,-176.372,8.648,148.665
C04443=1167.232,346.594,-77.473,-176.375,8.645,148.665
C04444=1167.236,346.347,-77.439,-176.377,8.642,148.665
C04445=1167.240,346.099,-77.406,-176.379,8.639,148.665
C04446=1167.244,345.851,-77.373,-176.382,8.634,148.665
C04447=1167.249,345.603,-77.339,-176.384,8.631,148.664
C04448=1167.253,345.356,-77.305,-176.387,8.628,148.664
C04449=1167.257,345.108,-77.272,-176.390,8.624,148.664
C04450=1167.260,344.860,-77.239,-176.392,8.620,148.664
C04451=1167.264,344.612,-77.205,-176.394,8.617,148.663
C04452=1167.269,344.364,-77.172,-176.396,8.614,148.663
C04453=1167.272,344.117,-77.138,-176.399,8.610,148.663
C04454=1167.277,343.870,-77.105,-176.402,8.606,148.663
C04455=1167.281,343.622,-77.072,-176.404,8.603,148.663
C04456=1167.285,343.374,-77.039,-176.406,8.600,148.662
C04457=1167.290,343.126,-77.005,-176.409,8.596,148.662
C04458=1167.294,342.878,-76.972,-176.411,8.592,148.662
C04459=1167.298,342.631,-76.939,-176.414,8.589,148.662
C04460=1167.302,342.382,-76.905,-176.416,8.586,148.661
C04461=1167.305,342.135,-76.872,-176.419,8.582,148.661
C04462=1167.310,341.887,-76.838,-176.421,8.578,148.661
C04463=1167.314,341.640,-76.805,-176.424,8.575,148.661
C04464=1167.318,341.392,-76.772,-176.426,8.572,148.661
C04465=1167.322,341.144,-76.739,-176.428,8.569,148.661
C04466=1167.326,340.896,-76.706,-176.431,8.565,148.660
C04467=1167.330,340.649,-76.673,-176.434,8.561,148.660
C04468=1167.334,340.401,-76.639,-176.436,8.558,148.660
C04469=1167.338,340.122,-76.602,-176.439,8.554,148.660
C04470=1167.343,339.842,-76.566,-176.442,8.550,148.659
C04471=1167.348,339.562,-76.528,-176.444,8.547,148.659
C04472=1167.353,339.283,-76.491,-176.447,8.542,148.659
C04473=1167.357,339.035,-76.458,-176.449,8.539,148.659
C04474=1167.361,338.788,-76.425,-176.452,8.535,148.659
C04475=1167.365,338.540,-76.392,-176.455,8.532,148.658
C04476=1167.369,338.292,-76.359,-176.457,8.529,148.658
C04477=1167.373,338.045,-76.326,-176.459,8.526,148.658
C04478=1167.377,337.796,-76.293,-176.462,8.521,148.658
C04479=1167.381,337.549,-76.260,-176.464,8.518,148.658
C04480=1167.386,337.301,-76.227,-176.467,8.515,148.657
C04481=1167.390,337.053,-76.194,-176.469,8.511,148.657
C04482=1167.394,336.805,-76.161,-176.472,8.509,148.657
C04483=1167.398,336.557,-76.129,-176.475,8.504,148.657
C04484=1167.402,336.310,-76.096,-176.477,8.501,148.657
C04485=1167.406,336.062,-76.063,-176.479,8.498,148.656
C04486=1167.410,335.814,-76.030,-176.481,8.495,148.656
C04487=1167.414,335.566,-75.998,-176.484,8.491,148.656
C04488=1167.418,335.318,-75.964,-176.487,8.487,148.656
C04489=1167.422,335.071,-75.931,-176.489,8.484,148.656
C04490=1167.426,334.822,-75.899,-176.492,8.481,148.656
C04491=1167.431,334.575,-75.866,-176.494,8.478,148.655
C04492=1167.434,334.327,-75.834,-176.496,8.474,148.655
C04493=1167.438,334.079,-75.801,-176.499,8.470,148.655
C04494=1167.443,333.831,-75.768,-176.502,8.467,148.655
C04495=1167.446,333.583,-75.736,-176.504,8.464,148.655
C04496=1167.451,333.336,-75.703,-176.506,8.461,148.655
C04497=1167.455,333.088,-75.670,-176.509,8.457,148.654
C04498=1167.459,332.840,-75.638,-176.511,8.454,148.654
C04499=1167.463,332.592,-75.605,-176.514,8.450,148.654
C04500=1167.467,332.344,-75.572,-176.517,8.447,148.654
C04501=1167.471,332.097,-75.540,-176.519,8.444,148.654
C04502=1167.475,331.848,-75.507,-176.521,8.440,148.653
C04503=1167.480,331.600,-75.475,-176.524,8.437,148.653
C04504=1167.484,331.353,-75.443,-176.527,8.433,148.653
C04505=1167.488,331.105,-75.410,-176.529,8.430,148.653
C04506=1167.492,330.857,-75.377,-176.531,8.427,148.653
C04507=1167.496,330.609,-75.345,-176.534,8.424,148.653
C04508=1167.500,330.362,-75.312,-176.536,8.420,148.653
C04509=1167.504,330.114,-75.280,-176.539,8.417,148.652
C04510=1167.508,329.865,-75.248,-176.541,8.413,148.652
C04511=1167.513,329.618,-75.215,-176.544,8.410,148.652
C04512=1167.517,329.370,-75.183,-176.546,8.407,148.652
C04513=1167.521,329.122,-75.150,-176.549,8.403,148.652
C04514=1167.525,328.874,-75.118,-176.551,8.400,148.652
C04515=1167.529,328.626,-75.086,-176.554,8.397,148.652
C04516=1167.533,328.379,-75.054,-176.556,8.394,148.651
C04517=1167.537,328.131,-75.021,-176.559,8.390,148.651
C04518=1167.541,327.883,-74.989,-176.562,8.387,148.651
C04519=1167.546,327.635,-74.957,-176.564,8.383,148.651
C04520=1167.550,327.388,-74.925,-176.566,8.380,148.651
C04521=1167.554,327.139,-74.892,-176.569,8.377,148.651
C04522=1167.558,326.891,-74.860,-176.571,8.374,148.651
C04523=1167.562,326.643,-74.828,-176.574,8.370,148.650
C04524=1167.566,326.395,-74.796,-176.576,8.366,148.650
C04525=1167.571,326.148,-74.763,-176.579,8.363,148.650
C04526=1167.574,325.900,-74.731,-176.581,8.360,148.650
C04527=1167.579,325.652,-74.699,-176.584,8.357,148.650
C04528=1167.583,325.404,-74.667,-176.586,8.354,148.650
C04529=1167.587,325.156,-74.636,-176.589,8.351,148.649
C04530=1167.591,324.908,-74.603,-176.592,8.346,148.649
C04531=1167.595,324.660,-74.571,-176.594,8.343,148.649
C04532=1167.600,324.412,-74.539,-176.597,8.340,148.649
C04533=1167.603,324.165,-74.507,-176.599,8.337,148.649
C04534=1167.607,323.917,-74.475,-176.602,8.334,148.649
C04535=1167.612,323.668,-74.442,-176.604,8.331,148.649
C04536=1167.616,323.421,-74.411,-176.606,8.327,148.648
C04537=1167.620,323.173,-74.379,-176.609,8.324,148.648
C04538=1167.624,322.925,-74.347,-176.612,8.320,148.648
C04539=1167.628,322.677,-74.315,-176.615,8.317,148.648
C04540=1167.632,322.429,-74.283,-176.617,8.314,148.648
C04541=1167.636,322.181,-74.251,-176.619,8.311,148.648
C04542=1167.641,321.934,-74.219,-176.622,8.308,148.648
C04543=1167.644,321.686,-74.188,-176.624,8.304,148.648
C04544=1167.648,321.437,-74.156,-176.626,8.301,148.647
C04545=1167.654,321.189,-74.124,-176.629,8.298,148.647
C04546=1167.657,320.941,-74.092,-176.632,8.294,148.647
C04547=1167.661,320.693,-74.061,-176.635,8.291,148.647
C04548=1167.665,320.446,-74.029,-176.637,8.288,148.647
C04549=1167.670,320.198,-73.997,-176.639,8.284,148.647
C04550=1167.673,319.949,-73.965,-176.642,8.281,148.647
C04551=1167.678,319.702,-73.933,-176.644,8.278,148.647
C04552=1167.682,319.453,-73.902,-176.647,8.275,148.647
C04553=1167.687,319.206,-73.870,-176.649,8.272,148.646
C04554=1167.690,318.958,-73.838,-176.652,8.269,148.646
C04555=1167.694,318.710,-73.806,-176.654,8.266,148.646
C04556=1167.699,318.462,-73.776,-176.657,8.261,148.646
C04557=1167.702,318.214,-73.744,-176.660,8.258,148.646
C04558=1167.707,317.966,-73.712,-176.662,8.255,148.646
C04559=1167.711,317.718,-73.680,-176.665,8.252,148.646
C04560=1167.716,317.470,-73.649,-176.667,8.249,148.646
C04561=1167.720,317.222,-73.617,-176.670,8.246,148.646
C04562=1167.723,316.974,-73.586,-176.672,8.243,148.646
C04563=1167.728,316.726,-73.555,-176.675,8.239,148.645
C04564=1167.732,316.478,-73.523,-176.677,8.236,148.645
C04565=1167.736,316.231,-73.491,-176.680,8.233,148.645
C04566=1167.740,315.982,-73.460,-176.682,8.230,148.645
C04567=1167.744,315.735,-73.429,-176.685,8.226,148.645
C04568=1167.749,315.486,-73.397,-176.688,8.223,148.645
C04569=1167.753,315.238,-73.366,-176.690,8.220,148.645
C04570=1167.757,314.990,-73.334,-176.693,8.217,148.645
C04571=1167.762,314.742,-73.303,-176.695,8.213,148.645
C04572=1167.765,314.494,-73.271,-176.698,8.210,148.645
C04573=1167.771,314.217,-73.237,-176.701,8.206,148.644
C04574=1167.775,313.940,-73.202,-176.704,8.203,148.644
C04575=1167.779,313.663,-73.166,-176.707,8.199,148.644
C04576=1167.784,313.386,-73.131,-176.709,8.196,148.644
C04577=1167.789,313.138,-73.100,-176.712,8.193,148.644
C04578=1167.792,312.890,-73.069,-176.714,8.190,148.644
C04579=1167.797,312.642,-73.038,-176.717,8.187,148.644
C04580=1167.801,312.394,-73.006,-176.719,8.184,148.644
C04581=1167.805,312.146,-72.975,-176.722,8.180,148.644
C04582=1167.810,311.898,-72.944,-176.725,8.177,148.644
C04583=1167.814,311.650,-72.913,-176.727,8.173,148.643
C04584=1167.817,311.402,-72.882,-176.730,8.170,148.643
C04585=1167.821,311.154,-72.851,-176.732,8.167,148.643
C04586=1167.826,310.906,-72.820,-176.735,8.164,148.643
C04587=1167.830,310.658,-72.789,-176.737,8.161,148.643
C04588=1167.834,310.410,-72.758,-176.740,8.158,148.643
C04589=1167.839,310.163,-72.726,-176.742,8.155,148.643
C04590=1167.843,309.914,-72.695,-176.745,8.152,148.643
C04591=1167.847,309.666,-72.664,-176.747,8.148,148.643
C04592=1167.851,309.418,-72.633,-176.750,8.145,148.643
C04593=1167.856,309.170,-72.602,-176.752,8.142,148.643
C04594=1167.859,308.922,-72.572,-176.755,8.139,148.643
C04595=1167.863,308.674,-72.541,-176.758,8.136,148.643
C04596=1167.868,308.426,-72.510,-176.760,8.133,148.642
C04597=1167.872,308.178,-72.478,-176.763,8.130,148.642
C04598=1167.876,307.930,-72.447,-176.765,8.126,148.642
C04599=1167.881,307.682,-72.416,-176.768,8.123,148.642
C04600=1167.884,307.433,-72.386,-176.771,8.119,148.642
C04601=1167.889,307.185,-72.355,-176.774,8.116,148.642
C04602=1167.894,306.937,-72.324,-176.776,8.113,148.642
C04603=1167.898,306.689,-72.293,-176.779,8.110,148.642
C04604=1167.902,306.441,-72.262,-176.781,8.107,148.642
C04605=1167.906,306.194,-72.232,-176.784,8.104,148.642
C04606=1167.910,305.945,-72.200,-176.786,8.101,148.642
C04607=1167.914,305.697,-72.170,-176.789,8.098,148.642
C04608=1167.919,305.449,-72.139,-176.791,8.095,148.642
C04609=1167.922,305.201,-72.108,-176.794,8.091,148.641
C04610=1167.927,304.953,-72.078,-176.796,8.088,148.641
C04611=1167.931,304.705,-72.047,-176.799,8.085,148.641
C04612=1167.935,304.457,-72.017,-176.801,8.082,148.641
C04613=1167.939,304.209,-71.986,-176.804,8.079,148.641
C04614=1167.944,303.961,-71.955,-176.806,8.076,148.641
C04615=1167.949,303.713,-71.924,-176.809,8.073,148.641
C04616=1167.952,303.465,-71.894,-176.812,8.070,148.641
C04617=1167.956,303.216,-71.863,-176.814,8.067,148.641
C04618=1167.961,302.968,-71.832,-176.817,8.064,148.641
C04619=1167.965,302.720,-71.803,-176.819,8.060,148.641
C04620=1167.970,302.472,-71.772,-176.822,8.057,148.641
C04621=1167.973,302.224,-71.741,-176.825,8.054,148.641
C04622=1167.978,301.976,-71.710,-176.827,8.051,148.641
C04623=1167.982,301.728,-71.680,-176.830,8.048,148.641
C04624=1167.986,301.480,-71.650,-176.832,8.045,148.641
C04625=1167.991,301.231,-71.619,-176.835,8.042,148.641
C04626=1167.994,300.983,-71.589,-176.838,8.039,148.641
C04627=1167.999,300.735,-71.558,-176.840,8.036,148.640
C04628=1168.004,300.487,-71.527,-176.843,8.033,148.640
C04629=1168.007,300.239,-71.497,-176.845,8.030,148.640
C04630=1168.012,299.991,-71.467,-176.848,8.026,148.640
C04631=1168.016,299.743,-71.437,-176.850,8.023,148.640
C04632=1168.020,299.495,-71.406,-176.853,8.020,148.640
C04633=1168.024,299.247,-71.376,-176.855,8.017,148.640
C04634=1168.029,298.999,-71.346,-176.858,8.014,148.640
C04635=1168.032,298.750,-71.315,-176.861,8.011,148.640
C04636=1168.037,298.502,-71.284,-176.863,8.008,148.640
C04637=1168.041,298.254,-71.255,-176.866,8.005,148.640
C04638=1168.046,298.006,-71.224,-176.869,8.002,148.640
C04639=1168.050,297.758,-71.195,-176.871,7.999,148.640
C04640=1168.055,297.510,-71.164,-176.874,7.996,148.640
C04641=1168.058,297.262,-71.133,-176.876,7.993,148.640
C04642=1168.063,297.013,-71.103,-176.879,7.989,148.640
C04643=1168.067,296.765,-71.073,-176.881,7.986,148.640
C04644=1168.071,296.517,-71.044,-176.884,7.983,148.640
C04645=1168.075,296.269,-71.013,-176.886,7.980,148.640
C04646=1168.079,296.022,-70.983,-176.889,7.977,148.640
C04647=1168.084,295.773,-70.953,-176.892,7.974,148.640
C04648=1168.088,295.525,-70.923,-176.894,7.971,148.639
C04649=1168.092,295.276,-70.893,-176.897,7.968,148.639
C04650=1168.096,295.028,-70.862,-176.900,7.965,148.640
C04651=1168.101,294.780,-70.833,-176.902,7.962,148.639
C04652=1168.105,294.532,-70.803,-176.905,7.959,148.639
C04653=1168.109,294.284,-70.772,-176.907,7.956,148.639
C04654=1168.113,294.036,-70.743,-176.910,7.953,148.639
C04655=1168.117,293.788,-70.713,-176.913,7.949,148.639
C04656=1168.122,293.539,-70.683,-176.915,7.946,148.639
C04657=1168.126,293.292,-70.653,-176.918,7.944,148.639
C04658=1168.130,293.043,-70.623,-176.920,7.940,148.639
C04659=1168.135,292.795,-70.593,-176.923,7.937,148.639
C04660=1168.139,292.547,-70.563,-176.926,7.934,148.639
C04661=1168.143,292.299,-70.533,-176.929,7.931,148.639
C04662=1168.148,292.051,-70.504,-176.931,7.928,148.639
C04663=1168.152,291.803,-70.473,-176.934,7.925,148.639
C04664=1168.156,291.554,-70.443,-176.936,7.922,148.639
C04665=1168.160,291.306,-70.414,-176.938,7.920,148.639
C04666=1168.164,291.057,-70.384,-176.941,7.917,148.639
C04667=1168.169,290.809,-70.354,-176.944,7.914,148.639
C04668=1168.173,290.561,-70.324,-176.946,7.911,148.639
C04669=1168.177,290.313,-70.295,-176.949,7.908,148.639
C04670=1168.181,290.064,-70.265,-176.951,7.904,148.639
C04671=1168.185,289.817,-70.235,-176.954,7.901,148.639
C04672=1168.190,289.568,-70.205,-176.957,7.898,148.639
C04673=1168.194,289.320,-70.176,-176.960,7.896,148.639
C04674=1168.199,289.072,-70.147,-176.962,7.892,148.639
C04675=1168.203,288.824,-70.117,-176.965,7.889,148.639
C04676=1168.207,288.576,-70.088,-176.967,7.886,148.639
C04677=1168.212,288.301,-70.054,-176.970,7.883,148.639
C04678=1168.217,288.026,-70.022,-176.973,7.880,148.639
C04679=1168.222,287.751,-69.988,-176.976,7.876,148.639
C04680=1168.226,287.476,-69.956,-176.978,7.873,148.639
C04681=1168.230,287.228,-69.927,-176.981,7.870,148.639
C04682=1168.235,286.979,-69.897,-176.984,7.867,148.639
C04683=1168.239,286.731,-69.867,-176.987,7.864,148.639
C04684=1168.244,286.483,-69.838,-176.989,7.861,148.639
C04685=1168.248,286.235,-69.809,-176.992,7.858,148.639
C04686=1168.252,285.987,-69.779,-176.994,7.855,148.639
C04687=1168.256,285.738,-69.750,-176.997,7.852,148.639
C04688=1168.261,285.490,-69.721,-177.000,7.849,148.639
C04689=1168.265,285.242,-69.691,-177.002,7.846,148.639
C04690=1168.269,284.994,-69.662,-177.005,7.843,148.639
C04691=1168.273,284.745,-69.632,-177.008,7.840,148.639
C04692=1168.277,284.497,-69.603,-177.010,7.838,148.639
C04693=1168.282,284.250,-69.574,-177.013,7.835,148.639
C04694=1168.286,284.001,-69.544,-177.015,7.832,148.639
C04695=1168.290,283.753,-69.515,-177.018,7.829,148.639
C04696=1168.295,283.505,-69.485,-177.020,7.826,148.639
C04697=1168.299,283.256,-69.456,-177.023,7.823,148.639
C04698=1168.303,283.008,-69.427,-177.026,7.820,148.639
C04699=1168.307,282.759,-69.398,-177.028,7.816,148.639
C04700=1168.312,282.512,-69.369,-177.031,7.813,148.639
C04701=1168.316,282.263,-69.339,-177.034,7.810,148.639
C04702=1168.321,282.015,-69.310,-177.036,7.807,148.639
C04703=1168.325,281.766,-69.281,-177.039,7.804,148.639
C04704=1168.329,281.518,-69.251,-177.041,7.802,148.639
C04705=1168.334,281.270,-69.222,-177.044,7.799,148.639
C04706=1168.338,281.023,-69.194,-177.046,7.796,148.639
C04707=1168.342,280.774,-69.165,-177.049,7.793,148.639
C04708=1168.346,280.525,-69.135,-177.052,7.790,148.639
C04709=1168.350,280.277,-69.106,-177.055,7.787,148.639
C04710=1168.355,280.029,-69.078,-177.057,7.784,148.639
C04711=1168.360,279.781,-69.048,-177.060,7.781,148.639
C04712=1168.364,279.532,-69.019,-177.062,7.778,148.639
C04713=1168.368,279.284,-68.990,-177.065,7.776,148.639
C04714=1168.372,279.036,-68.961,-177.067,7.773,148.639
C04715=1168.377,278.788,-68.932,-177.070,7.770,148.639
C04716=1168.381,278.539,-68.903,-177.073,7.767,148.639
C04717=1168.385,278.291,-68.874,-177.076,7.764,148.639
C04718=1168.389,278.042,-68.846,-177.078,7.761,148.639
C04719=1168.394,277.795,-68.817,-177.081,7.758,148.639
C04720=1168.398,277.546,-68.788,-177.083,7.755,148.639
C04721=1168.402,277.298,-68.758,-177.086,7.752,148.639
C04722=1168.407,277.050,-68.731,-177.088,7.750,148.639
C04723=1168.411,276.801,-68.701,-177.091,7.747,148.639
C04724=1168.415,276.552,-68.672,-177.094,7.744,148.639
C04725=1168.420,276.304,-68.643,-177.097,7.741,148.639
C04726=1168.424,276.056,-68.615,-177.099,7.738,148.639
C04727=1168.428,275.808,-68.586,-177.102,7.735,148.639
C04728=1168.433,275.559,-68.557,-177.105,7.732,148.639
C04729=1168.437,275.312,-68.528,-177.108,7.729,148.639
C04730=1168.441,275.063,-68.500,-177.109,7.726,148.639
C04731=1168.445,274.815,-68.470,-177.112,7.723,148.639
C04732=1168.450,274.567,-68.442,-177.115,7.720,148.639
C04733=1168.454,274.318,-68.414,-177.117,7.717,148.640
C04734=1168.458,274.070,-68.384,-177.120,7.715,148.640
C04735=1168.463,273.822,-68.356,-177.123,7.712,148.640
C04736=1168.467,273.573,-68.328,-177.126,7.709,148.640
C04737=1168.471,273.325,-68.298,-177.128,7.706,148.640
C04738=1168.476,273.077,-68.271,-177.131,7.703,148.640
C04739=1168.480,272.828,-68.242,-177.133,7.701,148.640
C04740=1168.484,272.580,-68.213,-177.136,7.698,148.640
C04741=1168.489,272.332,-68.185,-177.139,7.695,148.640
C04742=1168.493,272.083,-68.156,-177.142,7.692,148.640
C04743=1168.498,271.835,-68.128,-177.143,7.689,148.640
C04744=1168.502,271.587,-68.099,-177.146,7.686,148.640
C04745=1168.506,271.338,-68.070,-177.149,7.683,148.640
C04746=1168.511,271.090,-68.042,-177.152,7.680,148.640
C04747=1168.514,270.841,-68.014,-177.154,7.677,148.640
C04748=1168.519,270.593,-67.986,-177.157,7.674,148.640
C04749=1168.524,270.345,-67.956,-177.160,7.671,148.640
C04750=1168.527,270.096,-67.928,-177.162,7.669,148.640
C04751=1168.532,269.848,-67.900,-177.165,7.666,148.640
C04752=1168.536,269.600,-67.871,-177.168,7.663,148.640
C04753=1168.541,269.351,-67.843,-177.170,7.660,148.640
C04754=1168.545,269.103,-67.815,-177.173,7.657,148.640
C04755=1168.549,268.855,-67.787,-177.176,7.654,148.640
C04756=1168.554,268.606,-67.758,-177.178,7.652,148.641
C04757=1168.558,268.358,-67.731,-177.181,7.649,148.641
C04758=1168.563,268.109,-67.702,-177.183,7.646,148.641
C04759=1168.567,267.861,-67.674,-177.186,7.643,148.641
C04760=1168.571,267.613,-67.645,-177.189,7.640,148.641
C04761=1168.575,267.365,-67.617,-177.191,7.638,148.641
C04762=1168.580,267.116,-67.588,-177.194,7.635,148.641
C04763=1168.584,266.867,-67.561,-177.197,7.632,148.641
C04764=1168.588,266.619,-67.533,-177.199,7.629,148.641
C04765=1168.593,266.370,-67.504,-177.202,7.626,148.641
C04766=1168.597,266.123,-67.476,-177.205,7.623,148.641
C04767=1168.602,265.874,-67.448,-177.207,7.621,148.641
C04768=1168.606,265.626,-67.420,-177.210,7.618,148.641
C04769=1168.611,265.378,-67.392,-177.213,7.615,148.641
C04770=1168.615,265.129,-67.363,-177.215,7.612,148.641
C04771=1168.619,264.881,-67.336,-177.218,7.609,148.641
C04772=1168.623,264.633,-67.307,-177.220,7.607,148.641
C04773=1168.628,264.384,-67.279,-177.223,7.604,148.642
C04774=1168.632,264.135,-67.252,-177.226,7.601,148.642
C04775=1168.637,263.887,-67.224,-177.229,7.598,148.642
C04776=1168.641,263.638,-67.195,-177.231,7.595,148.642
C04777=1168.645,263.391,-67.167,-177.233,7.593,148.642
C04778=1168.650,263.143,-67.140,-177.236,7.590,148.642
C04779=1168.654,262.894,-67.112,-177.239,7.587,148.642
C04780=1168.659,262.645,-67.084,-177.242,7.584,148.642
C04781=1168.664,262.372,-67.053,-177.244,7.581,148.642
C04782=1168.668,262.099,-67.022,-177.248,7.579,148.642
C04783=1168.673,261.825,-66.992,-177.250,7.576,148.642
C04784=1168.678,261.553,-66.961,-177.253,7.573,148.642
C04785=1168.682,261.304,-66.933,-177.256,7.570,148.642
C04786=1168.686,261.056,-66.906,-177.259,7.567,148.642
C04787=1168.691,260.808,-66.878,-177.261,7.564,148.643
C04788=1168.695,260.559,-66.850,-177.264,7.562,148.643
C04789=1168.700,260.311,-66.822,-177.266,7.559,148.643
C04790=1168.704,260.062,-66.795,-177.269,7.556,148.643
C04791=1168.708,259.814,-66.767,-177.272,7.553,148.643
C04792=1168.713,259.566,-66.739,-177.275,7.550,148.643
C04793=1168.717,259.317,-66.712,-177.277,7.548,148.643
C04794=1168.722,259.069,-66.683,-177.280,7.545,148.643
C04795=1168.726,258.820,-66.656,-177.283,7.542,148.643
C04796=1168.730,258.572,-66.628,-177.286,7.539,148.643
C04797=1168.735,258.323,-66.601,-177.288,7.537,148.643
C04798=1168.739,258.075,-66.573,-177.290,7.534,148.644
C04799=1168.743,257.826,-66.546,-177.293,7.531,148.644
C04800=1168.748,257.578,-66.518,-177.296,7.528,148.644
C04801=1168.752,257.330,-66.491,-177.298,7.526,148.644
C04802=1168.756,257.081,-66.463,-177.301,7.523,148.644
C04803=1168.761,256.833,-66.436,-177.304,7.520,148.644
C04804=1168.765,256.585,-66.408,-177.307,7.518,148.644
C04805=1168.770,256.336,-66.380,-177.309,7.515,148.644
C04806=1168.774,256.087,-66.352,-177.312,7.513,148.644
C04807=1168.779,255.839,-66.325,-177.315,7.510,148.644
C04808=1168.783,255.590,-66.298,-177.317,7.507,148.644
C04809=1168.787,255.342,-66.270,-177.319,7.504,148.644
C04810=1168.792,255.093,-66.243,-177.322,7.502,148.645
C04811=1168.796,254.845,-66.215,-177.325,7.499,148.645
C04812=1168.801,254.597,-66.188,-177.328,7.496,148.645
C04813=1168.805,254.348,-66.161,-177.330,7.494,148.645
C04814=1168.809,254.100,-66.133,-177.333,7.491,148.645
C04815=1168.814,253.851,-66.106,-177.336,7.488,148.645
C04816=1168.819,253.603,-66.079,-177.339,7.485,148.645
C04817=1168.822,253.354,-66.052,-177.341,7.483,148.645
C04818=1168.826,253.106,-66.024,-177.344,7.480,148.645
C04819=1168.831,252.858,-65.997,-177.347,7.477,148.646
C04820=1168.835,252.609,-65.970,-177.349,7.475,148.646
C04821=1168.840,252.361,-65.943,-177.352,7.472,148.646
C04822=1168.844,252.112,-65.915,-177.355,7.469,148.646
C04823=1168.849,251.864,-65.888,-177.357,7.466,148.646
C04824=1168.853,251.615,-65.861,-177.359,7.464,148.646
C04825=1168.858,251.367,-65.834,-177.362,7.461,148.646
C04826=1168.863,251.118,-65.806,-177.365,7.458,148.646
C04827=1168.866,250.870,-65.779,-177.368,7.456,148.646
C04828=1168.870,250.621,-65.752,-177.370,7.453,148.646
C04829=1168.875,250.373,-65.725,-177.373,7.450,148.647
C04830=1168.880,250.124,-65.698,-177.376,7.447,148.647
C04831=1168.884,249.876,-65.671,-177.379,7.446,148.647
C04832=1168.889,249.627,-65.644,-177.381,7.443,148.647
C04833=1168.892,249.378,-65.617,-177.384,7.440,148.647
C04834=1168.897,249.130,-65.590,-177.386,7.438,148.647
C04835=1168.901,248.881,-65.563,-177.389,7.435,148.647
C04836=1168.906,248.633,-65.536,-177.392,7.432,148.647
C04837=1168.911,248.384,-65.509,-177.394,7.430,148.648
C04838=1168.915,248.136,-65.482,-177.397,7.427,148.648
C04839=1168.919,247.888,-65.455,-177.400,7.424,148.648
C04840=1168.924,247.639,-65.428,-177.403,7.421,148.648
C04841=1168.929,247.391,-65.401,-177.405,7.419,148.648
C04842=1168.932,247.142,-65.374,-177.408,7.416,148.648
C04843=1168.937,246.893,-65.347,-177.411,7.413,148.648
C04844=1168.941,246.645,-65.320,-177.413,7.411,148.648
C04845=1168.946,246.396,-65.293,-177.416,7.408,148.648
C04846=1168.950,246.148,-65.266,-177.419,7.406,148.649
C04847=1168.955,245.900,-65.239,-177.421,7.403,148.649
C04848=1168.959,245.651,-65.212,-177.424,7.400,148.649
C04849=1168.963,245.403,-65.186,-177.427,7.397,148.649
C04850=1168.968,245.154,-65.159,-177.429,7.396,148.649
C04851=1168.973,244.905,-65.132,-177.432,7.393,148.649
C04852=1168.977,244.657,-65.106,-177.435,7.390,148.649
C04853=1168.981,244.409,-65.079,-177.437,7.388,148.649
C04854=1168.986,244.160,-65.052,-177.440,7.385,148.650
C04855=1168.990,243.912,-65.025,-177.443,7.382,148.650
C04856=1168.995,243.663,-64.999,-177.445,7.380,148.650
C04857=1168.999,243.414,-64.972,-177.448,7.377,148.650
C04858=1169.003,243.166,-64.945,-177.451,7.374,148.650
C04859=1169.008,242.918,-64.918,-177.453,7.372,148.650
C04860=1169.012,242.669,-64.893,-177.456,7.369,148.650
C04861=1169.017,242.420,-64.866,-177.459,7.366,148.651
C04862=1169.021,242.172,-64.839,-177.462,7.365,148.651
C04863=1169.026,241.923,-64.813,-177.464,7.362,148.651
C04864=1169.030,241.675,-64.786,-177.467,7.359,148.651
C04865=1169.034,241.427,-64.759,-177.469,7.356,148.651
C04866=1169.039,241.177,-64.733,-177.472,7.354,148.651
C04867=1169.043,240.929,-64.706,-177.475,7.352,148.651
C04868=1169.048,240.681,-64.679,-177.477,7.349,148.652
C04869=1169.052,240.432,-64.654,-177.481,7.346,148.652
C04870=1169.057,240.183,-64.627,-177.483,7.344,148.652
C04871=1169.061,239.935,-64.600,-177.486,7.341,148.652
C04872=1169.066,239.686,-64.574,-177.488,7.338,148.652
C04873=1169.070,239.438,-64.547,-177.491,7.336,148.652
C04874=1169.075,239.189,-64.521,-177.494,7.333,148.652
C04875=1169.079,238.941,-64.494,-177.497,7.330,148.653
C04876=1169.083,238.692,-64.468,-177.499,7.329,148.653
C04877=1169.087,238.443,-64.442,-177.502,7.326,148.653
C04878=1169.092,238.194,-64.415,-177.504,7.323,148.653
C04879=1169.096,237.946,-64.389,-177.507,7.321,148.653
C04880=1169.100,237.697,-64.363,-177.510,7.318,148.653
C04881=1169.106,237.449,-64.336,-177.512,7.316,148.654
C04882=1169.110,237.201,-64.311,-177.516,7.313,148.654
C04883=1169.115,236.952,-64.284,-177.518,7.311,148.654
C04884=1169.119,236.703,-64.258,-177.520,7.308,148.654
C04885=1169.123,236.432,-64.229,-177.524,7.305,148.654
C04886=1169.129,236.160,-64.200,-177.526,7.303,148.654
C04887=1169.133,235.889,-64.172,-177.530,7.300,148.655
C04888=1169.138,235.616,-64.143,-177.532,7.297,148.655
C04889=1169.142,235.368,-64.117,-177.535,7.295,148.655
C04890=1169.147,235.119,-64.091,-177.538,7.292,148.655
C04891=1169.152,234.871,-64.065,-177.541,7.289,148.655
C04892=1169.156,234.623,-64.038,-177.543,7.287,148.655
C04893=1169.160,234.374,-64.013,-177.546,7.284,148.656
C04894=1169.165,234.125,-63.986,-177.548,7.282,148.656
C04895=1169.170,233.876,-63.961,-177.551,7.279,148.656
C04896=1169.173,233.628,-63.934,-177.554,7.277,148.656
C04897=1169.178,233.380,-63.909,-177.556,7.275,148.656
C04898=1169.183,233.131,-63.882,-177.560,7.272,148.656
C04899=1169.187,232.882,-63.856,-177.562,7.270,148.657
C04900=1169.191,232.634,-63.830,-177.565,7.267,148.657
C04901=1169.196,232.385,-63.804,-177.568,7.264,148.657
C04902=1169.201,232.136,-63.778,-177.570,7.262,148.657
C04903=1169.205,231.888,-63.753,-177.573,7.259,148.657
C04904=1169.210,231.639,-63.727,-177.575,7.257,148.657
C04905=1169.214,231.391,-63.700,-177.578,7.255,148.658
C04906=1169.219,231.142,-63.674,-177.581,7.253,148.658
C04907=1169.223,230.893,-63.649,-177.584,7.250,148.658
C04908=1169.228,230.645,-63.623,-177.586,7.247,148.658
C04909=1169.232,230.396,-63.597,-177.589,7.245,148.658
C04910=1169.237,230.148,-63.572,-177.592,7.242,148.658
C04911=1169.241,229.899,-63.546,-177.594,7.240,148.659
C04912=1169.246,229.650,-63.520,-177.597,7.237,148.659
C04913=1169.250,229.401,-63.494,-177.599,7.235,148.659
C04914=1169.255,229.153,-63.468,-177.603,7.233,148.659
C04915=1169.259,228.905,-63.442,-177.605,7.230,148.659
C04916=1169.263,228.656,-63.416,-177.608,7.228,148.660
C04917=1169.267,228.407,-63.391,-177.611,7.225,148.660
C04918=1169.272,228.159,-63.365,-177.613,7.223,148.660
C04919=1169.276,227.910,-63.339,-177.616,7.220,148.660
C04920=1169.281,227.661,-63.313,-177.618,7.218,148.660
C04921=1169.286,227.413,-63.288,-177.622,7.215,148.661
C04922=1169.291,227.163,-63.263,-177.624,7.213,148.661
C04923=1169.295,226.915,-63.237,-177.627,7.210,148.661
C04924=1169.300,226.667,-63.212,-177.629,7.209,148.661
C04925=1169.304,226.418,-63.186,-177.632,7.206,148.661
C04926=1169.308,226.169,-63.160,-177.635,7.204,148.662
C04927=1169.313,225.921,-63.135,-177.637,7.201,148.662
C04928=1169.317,225.672,-63.109,-177.640,7.199,148.662
C04929=1169.321,225.423,-63.083,-177.643,7.196,148.662
C04930=1169.326,225.175,-63.058,-177.646,7.193,148.662
C04931=1169.331,224.926,-63.033,-177.648,7.191,148.662
C04932=1169.335,224.677,-63.007,-177.651,7.188,148.662
C04933=1169.340,224.429,-62.982,-177.654,7.187,148.663
C04934=1169.344,224.180,-62.956,-177.656,7.184,148.663
C04935=1169.348,223.931,-62.930,-177.659,7.182,148.663
C04936=1169.353,223.682,-62.905,-177.662,7.179,148.663
C04937=1169.358,223.434,-62.880,-177.665,7.177,148.664
C04938=1169.362,223.186,-62.854,-177.667,7.174,148.664
C04939=1169.367,222.937,-62.829,-177.670,7.172,148.664
C04940=1169.371,222.687,-62.804,-177.673,7.169,148.664
C04941=1169.376,222.439,-62.778,-177.675,7.168,148.664
C04942=1169.380,222.190,-62.752,-177.678,7.165,148.665
C04943=1169.385,221.942,-62.728,-177.681,7.163,148.665
C04944=1169.389,221.693,-62.703,-177.684,7.160,148.665
C04945=1169.394,221.445,-62.677,-177.686,7.158,148.665
C04946=1169.398,221.196,-62.652,-177.689,7.155,148.665
C04947=1169.402,220.947,-62.626,-177.691,7.153,148.666
C04948=1169.407,220.699,-62.601,-177.694,7.150,148.666
C04949=1169.412,220.449,-62.576,-177.697,7.148,148.666
C04950=1169.416,220.202,-62.551,-177.700,7.146,148.666
C04951=1169.420,219.953,-62.525,-177.702,7.144,148.666
C04952=1169.425,219.704,-62.501,-177.705,7.141,148.667
C04953=1169.429,219.455,-62.475,-177.708,7.139,148.667
C04954=1169.435,219.207,-62.450,-177.711,7.136,148.667
C04955=1169.439,218.958,-62.425,-177.713,7.134,148.667
C04956=1169.443,218.709,-62.400,-177.716,7.132,148.668
C04957=1169.447,218.461,-62.375,-177.718,7.129,148.668
C04958=1169.452,218.211,-62.350,-177.721,7.128,148.668
C04959=1169.457,217.963,-62.324,-177.724,7.125,148.668
C04960=1169.461,217.714,-62.300,-177.726,7.123,148.668
C04961=1169.465,217.466,-62.275,-177.729,7.120,148.668
C04962=1169.470,217.216,-62.249,-177.732,7.118,148.669
C04963=1169.475,216.968,-62.224,-177.735,7.116,148.669
C04964=1169.479,216.720,-62.200,-177.737,7.113,148.669
C04965=1169.483,216.471,-62.174,-177.741,7.111,148.670
C04966=1169.488,216.222,-62.150,-177.743,7.109,148.670
C04967=1169.493,215.973,-62.125,-177.746,7.106,148.670
C04968=1169.497,215.725,-62.100,-177.748,7.104,148.670
C04969=1169.502,215.476,-62.075,-177.751,7.102,148.670
C04970=1169.507,215.227,-62.050,-177.754,7.099,148.671
C04971=1169.510,214.978,-62.025,-177.756,7.097,148.671
C04972=1169.515,214.730,-62.000,-177.759,7.094,148.671
C04973=1169.520,214.480,-61.975,-177.762,7.093,148.671
C04974=1169.524,214.232,-61.950,-177.764,7.090,148.671
C04975=1169.529,213.984,-61.926,-177.767,7.088,148.672
C04976=1169.534,213.734,-61.901,-177.770,7.085,148.672
C04977=1169.538,213.487,-61.876,-177.773,7.083,148.672
C04978=1169.542,213.237,-61.851,-177.775,7.081,148.673
C04979=1169.547,212.989,-61.827,-177.778,7.079,148.673
C04980=1169.552,212.740,-61.802,-177.781,7.077,148.673
C04981=1169.556,212.491,-61.776,-177.783,7.074,148.673
C04982=1169.560,212.243,-61.752,-177.786,7.072,148.673
C04983=1169.565,211.993,-61.727,-177.789,7.069,148.673
C04984=1169.569,211.745,-61.703,-177.792,7.067,148.674
C04985=1169.574,211.496,-61.679,-177.794,7.065,148.674
C04986=1169.578,211.248,-61.653,-177.797,7.063,148.674
C04987=1169.583,210.999,-61.629,-177.800,7.061,148.675
C04988=1169.588,210.750,-61.604,-177.802,7.058,148.675
C04989=1169.593,210.479,-61.577,-177.805,7.056,148.675
C04990=1169.597,210.210,-61.551,-177.808,7.053,148.675
C04991=1169.602,209.938,-61.524,-177.811,7.050,148.675
C04992=1169.607,209.668,-61.498,-177.814,7.048,148.676
C04993=1169.612,209.419,-61.473,-177.817,7.046,148.676
C04994=1169.616,209.170,-61.449,-177.819,7.044,148.676
C04995=1169.621,208.922,-61.423,-177.822,7.041,148.677
C04996=1169.625,208.674,-61.399,-177.825,7.039,148.677
C04997=1169.630,208.425,-61.375,-177.828,7.037,148.677
C04998=1169.634,208.176,-61.350,-177.831,7.035,148.677
C04999=1169.639,207.927,-61.325,-177.833,7.033,148.677
C05000=1169.644,207.679,-61.301,-177.836,7.030,148.678
C05001=1169.648,207.429,-61.276,-177.838,7.028,148.678
C05002=1169.653,207.181,-61.252,-177.841,7.025,148.678
C05003=1169.657,206.932,-61.229,-177.844,7.024,148.679
C05004=1169.663,206.683,-61.204,-177.846,7.022,148.679
C05005=1169.666,206.434,-61.180,-177.850,7.019,148.679
C05006=1169.671,206.185,-61.155,-177.852,7.017,148.679
C05007=1169.676,205.937,-61.131,-177.854,7.015,148.679
C05008=1169.680,205.688,-61.107,-177.858,7.012,148.680
C05009=1169.685,205.439,-61.082,-177.860,7.010,148.680
C05010=1169.689,205.190,-61.058,-177.863,7.008,148.680
C05011=1169.694,204.942,-61.033,-177.865,7.006,148.680
C05012=1169.699,204.693,-61.010,-177.868,7.004,148.681
C05013=1169.703,204.444,-60.985,-177.871,7.001,148.681
C05014=1169.708,204.195,-60.961,-177.873,6.999,148.681
C05015=1169.712,203.946,-60.937,-177.876,6.997,148.681
C05016=1169.717,203.698,-60.913,-177.879,6.995,148.682
C05017=1169.721,203.449,-60.888,-177.881,6.993,148.682
C05018=1169.726,203.200,-60.864,-177.885,6.990,148.682
C05019=1169.730,202.951,-60.840,-177.887,6.988,148.683
C05020=1169.735,202.703,-60.816,-177.890,6.986,148.683
C05021=1169.740,202.454,-60.791,-177.893,6.983,148.683
C05022=1169.744,202.204,-60.768,-177.895,6.981,148.683
C05023=1169.748,201.956,-60.744,-177.898,6.980,148.683
C05024=1169.753,201.707,-60.719,-177.901,6.977,148.684
C05025=1169.758,201.458,-60.696,-177.903,6.975,148.684
C05026=1169.763,201.210,-60.671,-177.906,6.973,148.684
C05027=1169.767,200.961,-60.647,-177.909,6.970,148.685
C05028=1169.771,200.712,-60.624,-177.911,6.968,148.685
C05029=1169.775,200.463,-60.600,-177.914,6.967,148.685
C05030=1169.781,200.214,-60.575,-177.917,6.964,148.685
C05031=1169.785,199.965,-60.552,-177.919,6.962,148.686
C05032=1169.790,199.717,-60.527,-177.922,6.960,148.686
C05033=1169.794,199.468,-60.504,-177.925,6.957,148.686
C05034=1169.799,199.220,-60.480,-177.928,6.955,148.686
C05035=1169.803,198.970,-60.455,-177.930,6.954,148.687
C05036=1169.808,198.721,-60.432,-177.933,6.951,148.687
C05037=1169.812,198.473,-60.408,-177.936,6.949,148.687
C05038=1169.817,198.224,-60.384,-177.938,6.947,148.687
C05039=1169.822,197.975,-60.360,-177.942,6.944,148.688
C05040=1169.826,197.726,-60.337,-177.944,6.942,148.688
C05041=1169.831,197.478,-60.313,-177.946,6.941,148.688
C05042=1169.835,197.229,-60.289,-177.950,6.938,148.689
C05043=1169.840,196.980,-60.265,-177.952,6.936,148.689
C05044=1169.845,196.731,-60.241,-177.955,6.934,148.689
C05045=1169.850,196.483,-60.217,-177.958,6.931,148.689
C05046=1169.854,196.233,-60.194,-177.960,6.929,148.690
C05047=1169.858,195.984,-60.169,-177.963,6.928,148.690
C05048=1169.863,195.735,-60.146,-177.966,6.925,148.690
C05049=1169.867,195.486,-60.123,-177.969,6.923,148.691
C05050=1169.872,195.238,-60.099,-177.971,6.921,148.691
C05051=1169.877,194.989,-60.075,-177.973,6.919,148.691
C05052=1169.881,194.741,-60.051,-177.977,6.917,148.691
C05053=1169.886,194.491,-60.028,-177.979,6.915,148.691
C05054=1169.890,194.242,-60.005,-177.982,6.913,148.692
C05055=1169.895,193.994,-59.980,-177.985,6.910,148.692
C05056=1169.899,193.745,-59.957,-177.988,6.908,148.693
C05057=1169.904,193.496,-59.934,-177.990,6.906,148.693
C05058=1169.909,193.247,-59.910,-177.993,6.904,148.693
C05059=1169.913,192.999,-59.886,-177.996,6.902,148.693
C05060=1169.918,192.749,-59.863,-177.998,6.900,148.693
C05061=1169.923,192.500,-59.840,-178.001,6.898,148.694
C05062=1169.927,192.252,-59.815,-178.004,6.896,148.694
C05063=1169.932,192.003,-59.792,-178.006,6.894,148.694
C05064=1169.936,191.754,-59.769,-178.009,6.892,148.695
C05065=1169.941,191.505,-59.745,-178.012,6.889,148.695
C05066=1169.946,191.256,-59.722,-178.015,6.887,148.695
C05067=1169.950,191.008,-59.698,-178.017,6.885,148.695
C05068=1169.954,190.759,-59.675,-178.019,6.883,148.696
C05069=1169.959,190.510,-59.652,-178.023,6.881,148.696
C05070=1169.964,190.261,-59.628,-178.025,6.879,148.696
C05071=1169.969,190.012,-59.605,-178.028,6.877,148.697
C05072=1169.974,189.763,-59.582,-178.030,6.875,148.697
C05073=1169.978,189.514,-59.559,-178.034,6.873,148.697
C05074=1169.983,189.266,-59.535,-178.036,6.871,148.698
C05075=1169.987,189.017,-59.511,-178.038,6.869,148.698
C05076=1169.991,188.768,-59.489,-178.041,6.867,148.698
C05077=1169.996,188.519,-59.465,-178.044,6.864,148.698
C05078=1170.001,188.270,-59.442,-178.047,6.863,148.699
C05079=1170.005,188.021,-59.419,-178.049,6.860,148.699
C05080=1170.010,187.772,-59.395,-178.052,6.859,148.699
C05081=1170.015,187.523,-59.372,-178.055,6.856,148.700
C05082=1170.019,187.275,-59.349,-178.058,6.854,148.700
C05083=1170.024,187.026,-59.326,-178.060,6.852,148.700
C05084=1170.029,186.777,-59.303,-178.063,6.850,148.700
C05085=1170.033,186.528,-59.279,-178.066,6.848,148.701
C05086=1170.037,186.279,-59.257,-178.069,6.846,148.701
C05087=1170.042,186.030,-59.233,-178.071,6.844,148.702
C05088=1170.047,185.781,-59.210,-178.073,6.842,148.702
C05089=1170.052,185.532,-59.186,-178.077,6.840,148.702
C05090=1170.056,185.284,-59.164,-178.079,6.838,148.702
C05091=1170.061,185.035,-59.141,-178.082,6.836,148.703
C05092=1170.066,184.786,-59.117,-178.084,6.834,148.703
C05093=1170.070,184.517,-59.093,-178.088,6.831,148.703
C05094=1170.075,184.247,-59.068,-178.090,6.830,148.704
C05095=1170.081,183.977,-59.043,-178.093,6.827,148.704
C05096=1170.085,183.708,-59.018,-178.096,6.825,148.704
C05097=1170.090,183.459,-58.995,-178.099,6.823,148.705
C05098=1170.095,183.209,-58.972,-178.102,6.821,148.705
C05099=1170.099,182.961,-58.949,-178.105,6.819,148.705
C05100=1170.104,182.712,-58.927,-178.107,6.817,148.705
C05101=1170.109,182.463,-58.903,-178.110,6.815,148.706
C05102=1170.113,182.214,-58.881,-178.113,6.813,148.706
C05103=1170.118,181.965,-58.857,-178.116,6.811,148.706
C05104=1170.123,181.715,-58.835,-178.118,6.809,148.707
C05105=1170.127,181.467,-58.812,-178.120,6.807,148.707
C05106=1170.132,181.218,-58.789,-178.123,6.805,148.707
C05107=1170.136,180.970,-58.766,-178.126,6.803,148.708
C05108=1170.141,180.720,-58.743,-178.129,6.801,148.708
C05109=1170.145,180.472,-58.721,-178.132,6.799,148.708
C05110=1170.150,180.223,-58.698,-178.134,6.797,148.709
C05111=1170.155,179.973,-58.675,-178.137,6.795,148.709
C05112=1170.159,179.725,-58.652,-178.140,6.793,148.709
C05113=1170.164,179.476,-58.629,-178.143,6.791,148.710
C05114=1170.169,179.227,-58.607,-178.145,6.789,148.710
C05115=1170.173,178.978,-58.584,-178.148,6.787,148.710
C05116=1170.177,178.729,-58.561,-178.150,6.785,148.710
C05117=1170.183,178.480,-58.539,-178.153,6.783,148.711
C05118=1170.187,178.231,-58.516,-178.156,6.781,148.711
C05119=1170.192,177.982,-58.493,-178.159,6.779,148.712
C05120=1170.196,177.734,-58.471,-178.161,6.777,148.712
C05121=1170.201,177.485,-58.448,-178.164,6.776,148.712
C05122=1170.205,177.235,-58.426,-178.166,6.773,148.712
C05123=1170.210,176.986,-58.402,-178.170,6.771,148.713
C05124=1170.215,176.738,-58.381,-178.172,6.769,148.713
C05125=1170.220,176.489,-58.357,-178.175,6.767,148.713
C05126=1170.224,176.239,-58.335,-178.178,6.766,148.714
C05127=1170.229,175.991,-58.313,-178.180,6.764,148.714
C05128=1170.234,175.742,-58.290,-178.183,6.762,148.715
C05129=1170.238,175.493,-58.267,-178.186,6.759,148.715
C05130=1170.243,175.244,-58.245,-178.189,6.757,148.715
C05131=1170.247,174.995,-58.222,-178.191,6.756,148.715
C05132=1170.253,174.746,-58.200,-178.194,6.754,148.716
C05133=1170.257,174.497,-58.178,-178.197,6.752,148.716
C05134=1170.261,174.248,-58.155,-178.199,6.750,148.717
C05135=1170.267,173.999,-58.133,-178.203,6.748,148.717
C05136=1170.270,173.751,-58.110,-178.205,6.746,148.717
C05137=1170.275,173.501,-58.088,-178.207,6.744,148.717
C05138=1170.280,173.252,-58.066,-178.210,6.742,148.718
C05139=1170.284,173.004,-58.043,-178.213,6.740,148.718
C05140=1170.289,172.755,-58.021,-178.215,6.739,148.718
C05141=1170.294,172.505,-57.999,-178.218,6.737,148.719
C05142=1170.298,172.257,-57.976,-178.221,6.734,148.719
C05143=1170.303,172.008,-57.954,-178.224,6.732,148.720
C05144=1170.308,171.758,-57.932,-178.226,6.730,148.720
C05145=1170.313,171.510,-57.909,-178.229,6.729,148.720
C05146=1170.317,171.261,-57.887,-178.232,6.727,148.720
C05147=1170.322,171.012,-57.865,-178.234,6.725,148.721
C05148=1170.327,170.763,-57.843,-178.237,6.723,148.721
C05149=1170.331,170.514,-57.820,-178.240,6.722,148.722
C05150=1170.336,170.265,-57.798,-178.243,6.719,148.722
C05151=1170.341,170.016,-57.776,-178.246,6.717,148.722
C05152=1170.345,169.767,-57.754,-178.248,6.715,148.723
C05153=1170.350,169.518,-57.732,-178.251,6.713,148.723
C05154=1170.354,169.270,-57.710,-178.253,6.712,148.723
C05155=1170.359,169.020,-57.687,-178.256,6.710,148.723
C05156=1170.364,168.771,-57.665,-178.259,6.708,148.724
C05157=1170.368,168.522,-57.643,-178.261,6.706,148.724
C05158=1170.373,168.273,-57.622,-178.265,6.704,148.725
C05159=1170.378,168.024,-57.599,-178.267,6.702,148.725
C05160=1170.383,167.775,-57.577,-178.270,6.700,148.725
C05161=1170.387,167.526,-57.554,-178.273,6.698,148.726
C05162=1170.392,167.278,-57.533,-178.275,6.697,148.726
C05163=1170.396,167.028,-57.511,-178.278,6.695,148.726
C05164=1170.401,166.780,-57.489,-178.280,6.693,148.727
C05165=1170.406,166.530,-57.466,-178.283,6.691,148.727
C05166=1170.411,166.281,-57.445,-178.286,6.689,148.727
C05167=1170.415,166.032,-57.423,-178.288,6.688,148.728
C05168=1170.420,165.783,-57.401,-178.292,6.685,148.728
C05169=1170.424,165.534,-57.379,-178.294,6.683,148.728
C05170=1170.429,165.285,-57.357,-178.297,6.681,148.729
C05171=1170.434,165.036,-57.335,-178.300,6.680,148.729
C05172=1170.438,164.787,-57.314,-178.302,6.678,148.729
C05173=1170.443,164.538,-57.291,-178.305,6.676,148.730
C05174=1170.448,164.289,-57.269,-178.308,6.674,148.730
C05175=1170.453,164.041,-57.248,-178.310,6.673,148.731
C05176=1170.457,163.791,-57.225,-178.313,6.671,148.731
C05177=1170.462,163.543,-57.204,-178.316,6.669,148.731
C05178=1170.467,163.293,-57.182,-178.318,6.667,148.731
C05179=1170.472,163.044,-57.161,-178.321,6.665,148.732
C05180=1170.476,162.795,-57.139,-178.324,6.663,148.732
C05181=1170.481,162.546,-57.117,-178.327,6.661,148.733
C05182=1170.486,162.297,-57.095,-178.329,6.659,148.733
C05183=1170.490,162.048,-57.073,-178.332,6.657,148.733
C05184=1170.495,161.799,-57.052,-178.335,6.656,148.734
C05185=1170.499,161.550,-57.030,-178.337,6.654,148.734
C05186=1170.504,161.301,-57.009,-178.340,6.652,148.734
C05187=1170.509,161.052,-56.987,-178.343,6.650,148.735
C05188=1170.513,160.803,-56.965,-178.345,6.649,148.735
C05189=1170.518,160.554,-56.943,-178.348,6.647,148.736
C05190=1170.523,160.305,-56.922,-178.351,6.645,148.736
C05191=1170.528,160.055,-56.900,-178.353,6.643,148.736
C05192=1170.533,159.807,-56.879,-178.356,6.642,148.737
C05193=1170.538,159.558,-56.857,-178.359,6.640,148.737
C05194=1170.541,159.309,-56.835,-178.362,6.638,148.737
C05195=1170.546,159.060,-56.814,-178.364,6.636,148.738
C05196=1170.551,158.811,-56.793,-178.367,6.635,148.738
C05197=1170.557,158.542,-56.769,-178.370,6.632,148.739
C05198=1170.561,158.274,-56.746,-178.373,6.630,148.739
C05199=1170.567,158.004,-56.723,-178.376,6.629,148.739
C05200=1170.571,157.735,-56.700,-178.379,6.626,148.740
C05201=1170.576,157.486,-56.678,-178.382,6.624,148.740
C05202=1170.581,157.236,-56.657,-178.384,6.622,148.740
C05203=1170.586,156.988,-56.635,-178.387,6.621,148.741
C05204=1170.590,156.739,-56.613,-178.390,6.619,148.741
C05205=1170.595,156.489,-56.592,-178.392,6.617,148.742
C05206=1170.599,156.241,-56.571,-178.395,6.615,148.742
C05207=1170.604,155.992,-56.550,-178.398,6.614,148.742
C05208=1170.609,155.743,-56.528,-178.400,6.612,148.743
C05209=1170.613,155.494,-56.506,-178.403,6.610,148.743
C05210=1170.619,155.244,-56.485,-178.406,6.608,148.743
C05211=1170.623,154.996,-56.464,-178.408,6.607,148.744
C05212=1170.628,154.747,-56.443,-178.411,6.605,148.744
C05213=1170.632,154.497,-56.421,-178.414,6.603,148.745
C05214=1170.637,154.248,-56.400,-178.417,6.601,148.745
C05215=1170.642,154.000,-56.379,-178.419,6.600,148.745
C05216=1170.647,153.751,-56.358,-178.422,6.598,148.746
C05217=1170.651,153.501,-56.336,-178.425,6.596,148.746
C05218=1170.656,153.252,-56.315,-178.427,6.594,148.746
C05219=1170.661,153.003,-56.293,-178.430,6.593,148.747
C05220=1170.665,152.754,-56.273,-178.433,6.591,148.747
C05221=1170.670,152.504,-56.252,-178.435,6.589,148.748
C05222=1170.675,152.256,-56.230,-178.438,6.587,148.748
C05223=1170.680,152.007,-56.209,-178.441,6.586,148.748
C05224=1170.684,151.758,-56.188,-178.443,6.584,148.749
C05225=1170.689,151.509,-56.167,-178.447,6.583,148.749
C05226=1170.695,151.260,-56.146,-178.449,6.581,148.750
C05227=1170.698,151.011,-56.125,-178.452,6.579,148.750
C05228=1170.703,150.761,-56.104,-178.455,6.577,148.750
C05229=1170.708,150.512,-56.083,-178.457,6.576,148.751
C05230=1170.713,150.264,-56.062,-178.460,6.574,148.751
C05231=1170.718,150.015,-56.041,-178.463,6.572,148.752
C05232=1170.723,149.765,-56.020,-178.466,6.570,148.752
C05233=1170.726,149.516,-55.998,-178.468,6.569,148.752
C05234=1170.732,149.267,-55.977,-178.471,6.567,148.753
C05235=1170.736,149.018,-55.957,-178.474,6.565,148.753
C05236=1170.741,148.769,-55.935,-178.476,6.563,148.753
C05237=1170.746,148.520,-55.914,-178.479,6.562,148.754
C05238=1170.751,148.271,-55.894,-178.482,6.560,148.754
C05239=1170.756,148.022,-55.873,-178.484,6.558,148.755
C05240=1170.760,147.772,-55.852,-178.487,6.556,148.755
C05241=1170.764,147.524,-55.831,-178.490,6.555,148.755
C05242=1170.770,147.274,-55.810,-178.492,6.554,148.756
C05243=1170.774,147.026,-55.789,-178.495,6.552,148.756
C05244=1170.779,146.776,-55.768,-178.497,6.550,148.757
C05245=1170.784,146.527,-55.748,-178.500,6.548,148.757
C05246=1170.788,146.279,-55.726,-178.503,6.547,148.757
C05247=1170.793,146.030,-55.706,-178.506,6.545,148.758
C05248=1170.798,145.780,-55.685,-178.509,6.544,148.758
C05249=1170.803,145.532,-55.664,-178.511,6.542,148.759
C05250=1170.807,145.282,-55.643,-178.514,6.540,148.759
C05251=1170.812,145.033,-55.623,-178.517,6.538,148.759
C05252=1170.817,144.783,-55.602,-178.519,6.537,148.760
C05253=1170.821,144.534,-55.581,-178.522,6.535,148.760
C05254=1170.826,144.285,-55.560,-178.525,6.533,148.761
C05255=1170.831,144.036,-55.540,-178.527,6.531,148.761
C05256=1170.836,143.787,-55.519,-178.530,6.530,148.761
C05257=1170.840,143.539,-55.498,-178.533,6.528,148.762
C05258=1170.845,143.289,-55.477,-178.536,6.526,148.762
C05259=1170.850,143.040,-55.457,-178.538,6.524,148.763
C05260=1170.854,142.791,-55.436,-178.541,6.523,148.763
C05261=1170.859,142.542,-55.415,-178.544,6.522,148.764
C05262=1170.864,142.293,-55.395,-178.546,6.520,148.764
C05263=1170.869,142.044,-55.374,-178.549,6.519,148.764
C05264=1170.874,141.794,-55.354,-178.552,6.517,148.765
C05265=1170.879,141.545,-55.333,-178.554,6.515,148.765
C05266=1170.883,141.296,-55.313,-178.557,6.513,148.765
C05267=1170.888,141.047,-55.293,-178.560,6.512,148.766
C05268=1170.893,140.798,-55.272,-178.562,6.510,148.766
C05269=1170.897,140.549,-55.251,-178.565,6.508,148.767
C05270=1170.902,140.300,-55.231,-178.568,6.506,148.767
C05271=1170.907,140.051,-55.210,-178.571,6.505,148.768
C05272=1170.911,139.802,-55.190,-178.574,6.503,148.768
C05273=1170.916,139.553,-55.169,-178.576,6.502,148.768
C05274=1170.921,139.303,-55.149,-178.579,6.501,148.769
C05275=1170.926,139.054,-55.129,-178.581,6.499,148.769
C05276=1170.930,138.805,-55.108,-178.584,6.497,148.770
C05277=1170.935,138.556,-55.087,-178.587,6.495,148.770
C05278=1170.940,138.307,-55.067,-178.589,6.494,148.770
C05279=1170.944,138.058,-55.046,-178.592,6.492,148.771
C05280=1170.950,137.808,-55.026,-178.595,6.490,148.771
C05281=1170.954,137.559,-55.006,-178.598,6.489,148.772
C05282=1170.959,137.310,-54.985,-178.601,6.487,148.772
C05283=1170.964,137.062,-54.965,-178.603,6.486,148.773
C05284=1170.969,136.812,-54.945,-178.605,6.484,148.773
C05285=1170.974,136.563,-54.925,-178.608,6.483,148.773
C05286=1170.978,136.314,-54.904,-178.611,6.481,148.774
C05287=1170.983,136.065,-54.885,-178.614,6.479,148.774
C05288=1170.988,135.815,-54.864,-178.617,6.478,148.775
C05289=1170.992,135.566,-54.844,-178.619,6.476,148.775
C05290=1170.997,135.317,-54.823,-178.622,6.474,148.775
C05291=1171.001,135.068,-54.803,-178.624,6.473,148.776
C05292=1171.007,134.820,-54.783,-178.627,6.472,148.776
C05293=1171.012,134.570,-54.763,-178.630,6.470,148.777
C05294=1171.016,134.321,-54.743,-178.632,6.468,148.777
C05295=1171.021,134.072,-54.722,-178.636,6.467,148.778
C05296=1171.026,133.822,-54.703,-178.638,6.465,148.778
C05297=1171.030,133.573,-54.682,-178.641,6.463,148.778
C05298=1171.034,133.324,-54.662,-178.644,6.462,148.779
C05299=1171.041,133.075,-54.642,-178.646,6.461,148.779
C05300=1171.045,132.826,-54.622,-178.648,6.459,148.780
C05301=1171.050,132.558,-54.601,-178.652,6.457,148.780
C05302=1171.056,132.289,-54.579,-178.654,6.456,148.781
C05303=1171.060,132.021,-54.557,-178.657,6.454,148.781
C05304=1171.066,131.752,-54.536,-178.661,6.452,148.782
C05305=1171.070,131.503,-54.515,-178.663,6.451,148.782
C05306=1171.075,131.253,-54.496,-178.666,6.449,148.782
C05307=1171.079,131.004,-54.475,-178.668,6.447,148.783
C05308=1171.084,130.755,-54.456,-178.671,6.446,148.783
C05309=1171.089,130.506,-54.436,-178.674,6.444,148.784
C05310=1171.094,130.257,-54.416,-178.677,6.443,148.784
C05311=1171.099,130.007,-54.396,-178.679,6.442,148.785
C05312=1171.103,129.758,-54.376,-178.682,6.440,148.785
C05313=1171.109,129.509,-54.357,-178.684,6.438,148.785
C05314=1171.113,129.260,-54.336,-178.687,6.436,148.786
C05315=1171.118,129.011,-54.316,-178.690,6.435,148.786
C05316=1171.122,128.762,-54.296,-178.693,6.433,148.787
C05317=1171.127,128.513,-54.277,-178.695,6.432,148.787
C05318=1171.132,128.264,-54.257,-178.698,6.431,148.788
C05319=1171.137,128.015,-54.237,-178.701,6.429,148.788
C05320=1171.141,127.765,-54.217,-178.703,6.427,148.788
C05321=1171.147,127.516,-54.198,-178.707,6.426,148.789
C05322=1171.151,127.267,-54.177,-178.709,6.424,148.789
C05323=1171.156,127.018,-54.158,-178.711,6.423,148.790
C05324=1171.161,126.768,-54.138,-178.714,6.421,148.790
C05325=1171.166,126.520,-54.118,-178.717,6.420,148.791
C05326=1171.170,126.270,-54.099,-178.719,6.418,148.791
C05327=1171.175,126.021,-54.079,-178.723,6.417,148.792
C05328=1171.180,125.771,-54.059,-178.725,6.415,148.792
C05329=1171.185,125.523,-54.039,-178.727,6.414,148.792
C05330=1171.190,125.273,-54.020,-178.730,6.412,148.793
C05331=1171.194,125.024,-54.000,-178.733,6.411,148.793
C05332=1171.200,124.775,-53.981,-178.736,6.409,148.794
C05333=1171.204,124.526,-53.960,-178.739,6.407,148.794
C05334=1171.208,124.277,-53.941,-178.741,6.406,148.795
C05335=1171.214,124.028,-53.922,-178.744,6.405,148.795
C05336=1171.218,123.778,-53.902,-178.746,6.403,148.795
C05337=1171.223,123.529,-53.883,-178.750,6.402,148.796
C05338=1171.228,123.280,-53.863,-178.752,6.400,148.796
C05339=1171.233,123.031,-53.843,-178.754,6.399,148.797
C05340=1171.238,122.781,-53.823,-178.757,6.397,148.797
C05341=1171.242,122.533,-53.805,-178.760,6.396,148.798
C05342=1171.247,122.283,-53.785,-178.763,6.394,148.798
C05343=1171.252,122.034,-53.765,-178.765,6.393,148.799
C05344=1171.257,121.785,-53.746,-178.768,6.392,148.799
C05345=1171.262,121.535,-53.726,-178.770,6.390,148.799
C05346=1171.267,121.286,-53.707,-178.774,6.388,148.800
C05347=1171.271,121.038,-53.687,-178.776,6.387,148.801
C05348=1171.276,120.788,-53.668,-178.779,6.386,148.801
C05349=1171.281,120.539,-53.648,-178.781,6.384,148.801
C05350=1171.286,120.290,-53.629,-178.784,6.382,148.802
C05351=1171.290,120.040,-53.610,-178.787,6.381,148.802
C05352=1171.295,119.792,-53.590,-178.789,6.380,148.803
C05353=1171.300,119.542,-53.571,-178.792,6.378,148.803
C05354=1171.305,119.293,-53.551,-178.795,6.377,148.804
C05355=1171.309,119.044,-53.532,-178.798,6.375,148.804
C05356=1171.314,118.794,-53.513,-178.800,6.374,148.805
C05357=1171.319,118.545,-53.493,-178.803,6.373,148.805
C05358=1171.324,118.296,-53.474,-178.805,6.371,148.805
C05359=1171.329,118.047,-53.455,-178.809,6.369,148.806
C05360=1171.334,117.797,-53.436,-178.811,6.368,148.806
C05361=1171.339,117.548,-53.417,-178.813,6.367,148.807
C05362=1171.343,117.299,-53.398,-178.816,6.365,148.807
C05363=1171.348,117.050,-53.378,-178.819,6.364,148.808
C05364=1171.353,116.800,-53.359,-178.822,6.362,148.808
C05365=1171.357,116.551,-53.340,-178.824,6.361,148.809
C05366=1171.362,116.302,-53.320,-178.827,6.359,148.809
C05367=1171.367,116.053,-53.301,-178.830,6.358,148.810
C05368=1171.372,115.804,-53.282,-178.833,6.356,148.810
C05369=1171.377,115.554,-53.263,-178.835,6.355,148.811
C05370=1171.382,115.305,-53.244,-178.838,6.354,148.811
C05371=1171.386,115.056,-53.225,-178.841,6.352,148.812
C05372=1171.391,114.807,-53.205,-178.843,6.351,148.812
C05373=1171.396,114.558,-53.186,-178.846,6.350,148.812
C05374=1171.401,114.308,-53.168,-178.848,6.348,148.813
C05375=1171.406,114.059,-53.148,-178.852,6.347,148.813
C05376=1171.410,113.810,-53.129,-178.854,6.346,148.814
C05377=1171.415,113.561,-53.110,-178.856,6.344,148.814
C05378=1171.421,113.311,-53.091,-178.859,6.342,148.815
C05379=1171.425,113.062,-53.072,-178.862,6.341,148.815
C05380=1171.430,112.813,-53.053,-178.864,6.340,148.816
C05381=1171.435,112.564,-53.034,-178.867,6.338,148.816
C05382=1171.440,112.314,-53.015,-178.870,6.336,148.816
C05383=1171.444,112.066,-52.997,-178.873,6.336,148.817
C05384=1171.449,111.816,-52.977,-178.875,6.334,148.818
C05385=1171.455,111.567,-52.958,-178.878,6.332,148.818
C05386=1171.459,111.317,-52.939,-178.881,6.331,148.819
C05387=1171.464,111.069,-52.920,-178.883,6.330,148.819
C05388=1171.469,110.819,-52.902,-178.886,6.328,148.819
C05389=1171.474,110.570,-52.882,-178.889,6.327,148.820
C05390=1171.478,110.321,-52.864,-178.891,6.326,148.820
C05391=1171.484,110.071,-52.845,-178.894,6.324,148.821
C05392=1171.488,109.823,-52.826,-178.897,6.323,148.821
C05393=1171.492,109.573,-52.808,-178.899,6.322,148.822
C05394=1171.498,109.324,-52.788,-178.902,6.320,148.822
C05395=1171.502,109.075,-52.770,-178.905,6.319,148.823
C05396=1171.507,108.825,-52.751,-178.907,6.317,148.823
C05397=1171.512,108.576,-52.732,-178.910,6.316,148.824
C05398=1171.517,108.326,-52.713,-178.913,6.315,148.824
C05399=1171.522,108.078,-52.694,-178.916,6.313,148.825
C05400=1171.527,107.828,-52.676,-178.918,6.313,148.825
C05401=1171.531,107.579,-52.657,-178.921,6.311,148.826
C05402=1171.536,107.330,-52.639,-178.924,6.309,148.826
C05403=1171.542,107.081,-52.619,-178.926,6.309,148.827
C05404=1171.546,106.831,-52.601,-178.929,6.307,148.827
C05405=1171.551,106.563,-52.580,-178.932,6.305,148.827
C05406=1171.557,106.295,-52.561,-178.935,6.304,148.828
C05407=1171.562,106.026,-52.541,-178.938,6.302,148.828
C05408=1171.566,105.758,-52.520,-178.941,6.301,148.829
C05409=1171.572,105.508,-52.502,-178.943,6.300,148.830
C05410=1171.576,105.259,-52.484,-178.946,6.298,148.830
C05411=1171.581,105.010,-52.465,-178.949,6.297,148.831
C05412=1171.587,104.761,-52.446,-178.951,6.296,148.831
C05413=1171.591,104.511,-52.427,-178.954,6.294,148.831
C05414=1171.596,104.262,-52.409,-178.957,6.293,148.832
C05415=1171.601,104.013,-52.391,-178.959,6.292,148.832
C05416=1171.606,103.764,-52.372,-178.962,6.290,148.833
C05417=1171.610,103.514,-52.354,-178.965,6.289,148.833
C05418=1171.616,103.265,-52.335,-178.967,6.288,148.834
C05419=1171.620,103.016,-52.316,-178.970,6.286,148.834
C05420=1171.625,102.766,-52.298,-178.973,6.285,148.835
C05421=1171.630,102.517,-52.280,-178.975,6.284,148.835
C05422=1171.635,102.268,-52.261,-178.978,6.282,148.836
C05423=1171.640,102.019,-52.243,-178.980,6.282,148.836
C05424=1171.644,101.769,-52.224,-178.983,6.280,148.837
C05425=1171.649,101.520,-52.206,-178.986,6.278,148.837
C05426=1171.655,101.271,-52.187,-178.988,6.278,148.838
C05427=1171.659,101.021,-52.169,-178.991,6.276,148.838
C05428=1171.664,100.772,-52.151,-178.994,6.274,148.839
C05429=1171.669,100.523,-52.133,-178.997,6.274,148.839
C05430=1171.674,100.274,-52.114,-178.999,6.272,148.840
C05431=1171.679,100.025,-52.096,-179.002,6.270,148.840
C05432=1171.683,99.775,-52.077,-179.005,6.270,148.841
C05433=1171.688,99.526,-52.059,-179.007,6.268,148.841
C05434=1171.693,99.277,-52.041,-179.010,6.266,148.842
C05435=1171.698,99.028,-52.022,-179.013,6.266,148.842
C05436=1171.703,98.778,-52.004,-179.015,6.264,148.843
C05437=1171.708,98.529,-51.986,-179.017,6.263,148.843
C05438=1171.713,98.280,-51.968,-179.021,6.262,148.844
C05439=1171.717,98.030,-51.950,-179.023,6.260,148.844
C05440=1171.722,97.781,-51.932,-179.026,6.259,148.845
C05441=1171.727,97.531,-51.913,-179.029,6.258,148.845
C05442=1171.732,97.282,-51.895,-179.031,6.257,148.846
C05443=1171.737,97.033,-51.877,-179.034,6.255,148.846
C05444=1171.742,96.784,-51.858,-179.037,6.254,148.847
C05445=1171.747,96.535,-51.840,-179.039,6.253,148.847
C05446=1171.752,96.286,-51.822,-179.042,6.251,148.848
C05447=1171.756,96.036,-51.804,-179.045,6.250,148.848
C05448=1171.761,95.787,-51.786,-179.047,6.249,148.849
C05449=1171.766,95.538,-51.768,-179.050,6.247,148.849
C05450=1171.771,95.288,-51.750,-179.052,6.247,148.850
C05451=1171.776,95.039,-51.732,-179.055,6.245,148.850
C05452=1171.781,94.790,-51.714,-179.058,6.244,148.851
C05453=1171.786,94.540,-51.695,-179.060,6.243,148.851
C05454=1171.790,94.291,-51.677,-179.063,6.241,148.852
C05455=1171.795,94.041,-51.659,-179.066,6.240,148.852
C05456=1171.800,93.792,-51.641,-179.068,6.239,148.853
C05457=1171.805,93.543,-51.623,-179.071,6.237,148.853
C05458=1171.810,93.293,-51.606,-179.074,6.236,148.854
C05459=1171.815,93.044,-51.588,-179.077,6.235,148.854
C05460=1171.820,92.795,-51.570,-179.079,6.234,148.855
C05461=1171.825,92.546,-51.552,-179.082,6.233,148.855
C05462=1171.829,92.296,-51.534,-179.084,6.232,148.856
C05463=1171.834,92.047,-51.516,-179.087,6.230,148.856
C05464=1171.839,91.798,-51.498,-179.090,6.229,148.857
C05465=1171.844,91.548,-51.480,-179.092,6.228,148.857
C05466=1171.849,91.299,-51.462,-179.095,6.226,148.858
C05467=1171.854,91.049,-51.444,-179.097,6.225,148.858
C05468=1171.859,90.801,-51.427,-179.101,6.224,148.859
C05469=1171.863,90.551,-51.409,-179.103,6.223,148.859
C05470=1171.868,90.302,-51.391,-179.105,6.221,148.860
C05471=1171.873,90.053,-51.373,-179.109,6.220,148.860
C05472=1171.878,89.803,-51.356,-179.111,6.219,148.861
C05473=1171.883,89.554,-51.338,-179.114,6.218,148.861
C05474=1171.888,89.305,-51.320,-179.116,6.217,148.862
C05475=1171.893,89.056,-51.302,-179.119,6.215,148.862
C05476=1171.898,88.807,-51.284,-179.122,6.215,148.863
C05477=1171.903,88.556,-51.266,-179.124,6.213,148.863
C05478=1171.908,88.307,-51.248,-179.127,6.211,148.864
